LIN {X 0,Y 607.534,Z 521.411,A -85,B 0,C 180,E1 27658.35,E2 27658.35} C_VEL
LIN {X 0,Y 606.937,Z 539.809,A -85,B 0,C 180,E1 27658.034,E2 27658.034} C_VEL
LIN {X 0,Y 606.179,Z 557.221,A -85,B 0,C 180,E1 27657.624,E2 27657.624} C_VEL
LIN {X 0,Y 605.306,Z 574.046,A -85,B 0,C 180,E1 27657.12,E2 27657.12} C_VEL
LIN {X 0,Y 604.323,Z 590.19,A -85,B 0,C 180,E1 27656.53,E2 27656.53} C_VEL
LIN {X 0,Y 603.193,Z 607.046,A -85,B 0,C 180,E1 27655.795,E2 27655.795} C_VEL
LIN {X 0,Y 601.778,Z 626.286,A -85,B 0,C 180,E1 27654.802,E2 27654.802} C_VEL
LIN {X 0,Y 600.164,Z 646.019,A -85,B 0,C 180,E1 27653.565,E2 27653.565} C_VEL
LIN {X 0,Y 598.909,Z 660.987,A -85,B 0,C 180,E1 27652.474,E2 27652.474} C_VEL
LIN {X 0,Y 597.728,Z 674.768,A -85,B 0,C 180,E1 27651.333,E2 27651.333} C_VEL
LIN {X 0,Y 596.656,Z 687.506,A -85,B 0,C 180,E1 27650.141,E2 27650.141} C_VEL
LIN {X 0,Y 595.699,Z 699.296,A -85,B 0,C 180,E1 27648.899,E2 27648.899} C_VEL
LIN {X 0,Y 594.784,Z 710.992,A -85,B 0,C 180,E1 27647.51,E2 27647.51} C_VEL
LIN {X 0,Y 593.947,Z 722.712,A -85,B 0,C 180,E1 27645.924,E2 27645.924} C_VEL
LIN {X 0,Y 593.118,Z 735.863,A -85,B 0,C 180,E1 27643.823,E2 27643.823} C_VEL
LIN {X 0,Y 592.654,Z 744.533,A -85,B 0,C 180,E1 27642.173,E2 27642.173} C_VEL
LIN {X 0,Y 592.352,Z 751.606,A -85,B 0,C 180,E1 27640.601,E2 27640.601} C_VEL
LIN {X 0,Y 592.127,Z 757.906,A -85,B 0,C 180,E1 27638.936,E2 27638.936} C_VEL
LIN {X 0,Y 592.011,Z 763.04,A -85,B 0,C 180,E1 27637.276,E2 27637.276} C_VEL
LIN {X 0,Y 591.947,Z 767.067,A -85,B 0,C 180,E1 27635.622,E2 27635.622} C_VEL
LIN {X 0,Y 591.925,Z 770.029,A -85,B 0,C 180,E1 27633.971,E2 27633.971} C_VEL
LIN {X 0,Y 591.913,Z 772.046,A -85,B 0,C 180,E1 27632.226,E2 27632.226} C_VEL
LIN {X 0,Y 591.908,Z 772.99,A -85,B 0,C 180,E1 27630.29,E2 27630.29} C_VEL
LIN {X 0,Y 591.917,Z 772.222,A -85,B 0,C 180,E1 27627.967,E2 27627.967} C_VEL
LIN {X 0,Y 591.924,Z 770.176,A -85,B 0,C 180,E1 27626.126,E2 27626.126} C_VEL
LIN {X 0,Y 591.944,Z 767.274,A -85,B 0,C 180,E1 27624.476,E2 27624.476} C_VEL
LIN {X 0,Y 592.002,Z 763.31,A -85,B 0,C 180,E1 27622.821,E2 27622.821} C_VEL
LIN {X 0,Y 592.116,Z 758.239,A -85,B 0,C 180,E1 27621.162,E2 27621.162} C_VEL
LIN {X 0,Y 592.323,Z 752.405,A -85,B 0,C 180,E1 27619.595,E2 27619.595} C_VEL
LIN {X 0,Y 592.61,Z 745.469,A -85,B 0,C 180,E1 27618.024,E2 27618.024} C_VEL
LIN {X 0,Y 593.024,Z 737.35,A -85,B 0,C 180,E1 27616.448,E2 27616.448} C_VEL
LIN {X 0,Y 593.643,Z 727.32,A -85,B 0,C 180,E1 27614.769,E2 27614.769} C_VEL
LIN {X 0,Y 594.627,Z 713.225,A -85,B 0,C 180,E1 27612.77,E2 27612.77} C_VEL
LIN {X 0,Y 595.607,Z 700.484,A -85,B 0,C 180,E1 27611.233,E2 27611.233} C_VEL
LIN {X 0,Y 596.616,Z 688.006,A -85,B 0,C 180,E1 27609.909,E2 27609.909} C_VEL
LIN {X 0,Y 597.677,Z 675.329,A -85,B 0,C 180,E1 27608.717,E2 27608.717} C_VEL
LIN {X 0,Y 598.853,Z 661.617,A -85,B 0,C 180,E1 27607.575,E2 27607.575} C_VEL
LIN {X 0,Y 600.104,Z 646.73,A -85,B 0,C 180,E1 27606.484,E2 27606.484} C_VEL
LIN {X 0,Y 601.642,Z 628.036,A -85,B 0,C 180,E1 27605.297,E2 27605.297} C_VEL
LIN {X 0,Y 603.118,Z 608.215,A -85,B 0,C 180,E1 27604.259,E2 27604.259} C_VEL
LIN {X 0,Y 604.251,Z 591.435,A -85,B 0,C 180,E1 27603.519,E2 27603.519} C_VEL
LIN {X 0,Y 605.262,Z 574.876,A -85,B 0,C 180,E1 27602.908,E2 27602.908} C_VEL
LIN {X 0,Y 606.173,Z 557.347,A -85,B 0,C 180,E1 27602.379,E2 27602.379} C_VEL
LIN {X 0,Y 606.929,Z 539.917,A -85,B 0,C 180,E1 27601.968,E2 27601.968} C_VEL
LIN {X 0,Y 607.522,Z 521.806,A -85,B 0,C 180,E1 27601.656,E2 27601.656} C_VEL
LIN {X 0,Y 611.396,Z 259.873,A -85,B 0,C 180,E1 27598.361,E2 27598.361} C_VEL
LIN {X 0,Y 611.12,Z 255.681,A -85,B 0,C 180,E1 27598.289,E2 27598.289} C_VEL
LIN {X 0,Y 604.007,Z 223.457,A -85,B 0,C 180,E1 27597.418,E2 27597.418} C_VEL
LIN {X 0,Y 601.164,Z 213.241,A -85,B 0,C 180,E1 27596.258,E2 27596.258} C_VEL
LIN {X 0,Y 594.896,Z 192.872,A -85,B 0,C 180,E1 27593.782,E2 27593.782} C_VEL
LIN {X 0,Y 593.129,Z 187.4,A -85,B 0,C 180,E1 27593.041,E2 27593.041} C_VEL
LIN {X 0,Y 593.122,Z 187.284,A -85,B 0,C 180,E1 27589.917,E2 27589.917} C_VEL
LIN {X 0,Y 593.118,Z 187.278,A -85,B 0,C 180,E1 27587.025,E2 27587.025} C_VEL
LIN {X 0,Y 593.105,Z 187.276,A -85,B 0,C 180,E1 27583.726,E2 27583.726} C_VEL
LIN {X 0,Y 593.165,Z 187.265,A -85,B 0,C 180,E1 27580.672,E2 27580.672} C_VEL
LIN {X 0,Y 593.102,Z 187.286,A -85,B 0,C 180,E1 27577.604,E2 27577.604} C_VEL
LIN {X 0,Y 593.164,Z 187.259,A -85,B 0,C 180,E1 27574.494,E2 27574.494} C_VEL
LIN {X 0,Y 593.104,Z 187.285,A -85,B 0,C 180,E1 27571.468,E2 27571.468} C_VEL
LIN {X 0,Y 593.129,Z 187.242,A -85,B 0,C 180,E1 27568.275,E2 27568.275} C_VEL
LIN {X 0,Y 593.113,Z 187.278,A -85,B 0,C 180,E1 27565.354,E2 27565.354} C_VEL
LIN {X 0,Y 593.109,Z 187.274,A -85,B 0,C 180,E1 27562.083,E2 27562.083} C_VEL
LIN {X 0,Y 593.131,Z 187.283,A -85,B 0,C 180,E1 27559.192,E2 27559.192} C_VEL
LIN {X 0,Y 593.106,Z 187.282,A -85,B 0,C 180,E1 27556.05,E2 27556.05} C_VEL
LIN {X 0,Y 593.141,Z 187.272,A -85,B 0,C 180,E1 27553.155,E2 27553.155} C_VEL
LIN {X 0,Y 593.102,Z 187.282,A -85,B 0,C 180,E1 27550,E2 27550} C_VEL
LIN {X 0,Y 593.178,Z 187.272,A -85,B 0,C 180,E1 27546.874,E2 27546.874} C_VEL
LIN {X 0,Y 593.101,Z 187.279,A -85,B 0,C 180,E1 27543.77,E2 27543.77} C_VEL
LIN {X 0,Y 593.129,Z 187.285,A -85,B 0,C 180,E1 27540.58,E2 27540.58} C_VEL
LIN {X 0,Y 593.107,Z 187.271,A -85,B 0,C 180,E1 27537.681,E2 27537.681} C_VEL
LIN {X 0,Y 593.108,Z 187.281,A -85,B 0,C 180,E1 27534.389,E2 27534.389} C_VEL
LIN {X 0,Y 593.122,Z 187.277,A -85,B 0,C 180,E1 27531.566,E2 27531.566} C_VEL
LIN {X 0,Y 593.102,Z 187.274,A -85,B 0,C 180,E1 27528.328,E2 27528.328} C_VEL
LIN {X 0,Y 593.169,Z 187.284,A -85,B 0,C 180,E1 27525.254,E2 27525.254} C_VEL
LIN {X 0,Y 593.101,Z 187.279,A -85,B 0,C 180,E1 27522.132,E2 27522.132} C_VEL
LIN {X 0,Y 593.154,Z 187.272,A -85,B 0,C 180,E1 27519.028,E2 27519.028} C_VEL
LIN {X 0,Y 593.102,Z 187.285,A -85,B 0,C 180,E1 27516.133,E2 27516.133} C_VEL
LIN {X 0,Y 593.144,Z 187.24,A -85,B 0,C 180,E1 27513.034,E2 27513.034} C_VEL
LIN {X 0,Y 593.105,Z 187.274,A -85,B 0,C 180,E1 27510.044,E2 27510.044} C_VEL
LIN {X 0,Y 593.11,Z 187.273,A -85,B 0,C 180,E1 27506.727,E2 27506.727} C_VEL
LIN {X 0,Y 593.135,Z 187.257,A -85,B 0,C 180,E1 27503.722,E2 27503.722} C_VEL
LIN {X 0,Y 593.104,Z 187.286,A -85,B 0,C 180,E1 27500.663,E2 27500.663} C_VEL
LIN {X 0,Y 593.148,Z 187.286,A -85,B 0,C 180,E1 27497.726,E2 27497.726} C_VEL
LIN {X 0,Y 593.101,Z 187.287,A -85,B 0,C 180,E1 27494.648,E2 27494.648} C_VEL
LIN {X 0,Y 593.18,Z 187.282,A -85,B 0,C 180,E1 27491.545,E2 27491.545} C_VEL
LIN {X 0,Y 593.099,Z 187.287,A -85,B 0,C 180,E1 27488.533,E2 27488.533} C_VEL
LIN {X 0,Y 593.16,Z 187.283,A -85,B 0,C 180,E1 27485.437,E2 27485.437} C_VEL
LIN {X 0,Y 593.104,Z 187.288,A -85,B 0,C 180,E1 27482.414,E2 27482.414} C_VEL
LIN {X 0,Y 593.12,Z 187.288,A -85,B 0,C 180,E1 27479.152,E2 27479.152} C_VEL
LIN {X 0,Y 593.123,Z 187.285,A -85,B 0,C 180,E1 27476.207,E2 27476.207} C_VEL
LIN {X 0,Y 593.105,Z 187.288,A -85,B 0,C 180,E1 27474.901,E2 27474.901} C_VEL
LIN {X 0,Y 592.123,Z 187.413,A -85,B 0,C 180,E1 27474.158,E2 27474.158} C_VEL
LIN {X 0,Y 585.692,Z 188.216,A -85,B 0,C 180,E1 27472.015,E2 27472.015} C_VEL
LIN {X 0,Y 585.212,Z 188.273,A -85,B 0,C 180,E1 27471.526,E2 27471.526} C_VEL
LIN {X 0,Y 585.169,Z 188.277,A -85,B 0,C 180,E1 27468.496,E2 27468.496} C_VEL
LIN {X 0,Y 585.169,Z 188.279,A -85,B 0,C 180,E1 27465.153,E2 27465.153} C_VEL
LIN {X 0,Y 585.197,Z 188.276,A -85,B 0,C 180,E1 27462.219,E2 27462.219} C_VEL
LIN {X 0,Y 585.16,Z 188.277,A -85,B 0,C 180,E1 27459.011,E2 27459.011} C_VEL
LIN {X 0,Y 585.234,Z 188.269,A -85,B 0,C 180,E1 27455.981,E2 27455.981} C_VEL
LIN {X 0,Y 585.161,Z 188.279,A -85,B 0,C 180,E1 27452.84,E2 27452.84} C_VEL
LIN {X 0,Y 585.19,Z 188.274,A -85,B 0,C 180,E1 27449.608,E2 27449.608} C_VEL
LIN {X 0,Y 585.171,Z 188.276,A -85,B 0,C 180,E1 27446.67,E2 27446.67} C_VEL
LIN {X 0,Y 585.166,Z 188.28,A -85,B 0,C 180,E1 27443.328,E2 27443.328} C_VEL
LIN {X 0,Y 585.208,Z 188.275,A -85,B 0,C 180,E1 27440.357,E2 27440.357} C_VEL
LIN {X 0,Y 585.161,Z 188.276,A -85,B 0,C 180,E1 27437.268,E2 27437.268} C_VEL
LIN {X 0,Y 585.233,Z 188.27,A -85,B 0,C 180,E1 27434.239,E2 27434.239} C_VEL
LIN {X 0,Y 585.162,Z 188.278,A -85,B 0,C 180,E1 27431.161,E2 27431.161} C_VEL
LIN {X 0,Y 585.213,Z 188.273,A -85,B 0,C 180,E1 27428.029,E2 27428.029} C_VEL
LIN {X 0,Y 585.168,Z 188.278,A -85,B 0,C 180,E1 27425.039,E2 27425.039} C_VEL
LIN {X 0,Y 585.177,Z 188.277,A -85,B 0,C 180,E1 27421.755,E2 27421.755} C_VEL
LIN {X 0,Y 585.185,Z 188.274,A -85,B 0,C 180,E1 27418.825,E2 27418.825} C_VEL
LIN {X 0,Y 585.164,Z 188.277,A -85,B 0,C 180,E1 27415.562,E2 27415.562} C_VEL
LIN {X 0,Y 585.234,Z 188.271,A -85,B 0,C 180,E1 27412.421,E2 27412.421} C_VEL
LIN {X 0,Y 585.163,Z 188.275,A -85,B 0,C 180,E1 27409.348,E2 27409.348} C_VEL
LIN {X 0,Y 585.207,Z 188.274,A -85,B 0,C 180,E1 27406.22,E2 27406.22} C_VEL
LIN {X 0,Y 585.173,Z 188.276,A -85,B 0,C 180,E1 27403.154,E2 27403.154} C_VEL
LIN {X 0,Y 585.168,Z 188.275,A -85,B 0,C 180,E1 27399.85,E2 27399.85} C_VEL
LIN {X 0,Y 585.198,Z 188.259,A -85,B 0,C 180,E1 27396.915,E2 27396.915} C_VEL
LIN {X 0,Y 585.16,Z 188.26,A -85,B 0,C 180,E1 27393.734,E2 27393.734} C_VEL
LIN {X 0,Y 585.239,Z 188.262,A -85,B 0,C 180,E1 27390.607,E2 27390.607} C_VEL
LIN {X 0,Y 585.16,Z 188.225,A -85,B 0,C 180,E1 27387.475,E2 27387.475} C_VEL
LIN {X 0,Y 585.178,Z 188.274,A -85,B 0,C 180,E1 27384.173,E2 27384.173} C_VEL
LIN {X 0,Y 585.177,Z 188.262,A -85,B 0,C 180,E1 27381.343,E2 27381.343} C_VEL
LIN {X 0,Y 585.17,Z 188.267,A -85,B 0,C 180,E1 27378.119,E2 27378.119} C_VEL
LIN {X 0,Y 585.212,Z 188.269,A -85,B 0,C 180,E1 27375.053,E2 27375.053} C_VEL
LIN {X 0,Y 585.16,Z 188.261,A -85,B 0,C 180,E1 27371.932,E2 27371.932} C_VEL
LIN {X 0,Y 585.231,Z 188.265,A -85,B 0,C 180,E1 27368.845,E2 27368.845} C_VEL
LIN {X 0,Y 585.163,Z 188.27,A -85,B 0,C 180,E1 27365.786,E2 27365.786} C_VEL
LIN {X 0,Y 585.187,Z 188.258,A -85,B 0,C 180,E1 27362.546,E2 27362.546} C_VEL
LIN {X 0,Y 585.174,Z 188.273,A -85,B 0,C 180,E1 27359.608,E2 27359.608} C_VEL
LIN {X 0,Y 585.164,Z 188.266,A -85,B 0,C 180,E1 27356.277,E2 27356.277} C_VEL
LIN {X 0,Y 585.237,Z 188.259,A -85,B 0,C 180,E1 27353.131,E2 27353.131} C_VEL
LIN {X 0,Y 585.162,Z 188.271,A -85,B 0,C 180,E1 27350.062,E2 27350.062} C_VEL
LIN {X 0,Y 585.204,Z 188.262,A -85,B 0,C 180,E1 27346.85,E2 27346.85} C_VEL
LIN {X 0,Y 585.168,Z 188.273,A -85,B 0,C 180,E1 27343.93,E2 27343.93} C_VEL
LIN {X 0,Y 585.173,Z 188.274,A -85,B 0,C 180,E1 27340.575,E2 27340.575} C_VEL
LIN {X 0,Y 585.203,Z 188.261,A -85,B 0,C 180,E1 27337.553,E2 27337.553} C_VEL
LIN {X 0,Y 585.164,Z 188.267,A -85,B 0,C 180,E1 27334.386,E2 27334.386} C_VEL
LIN {X 0,Y 585.234,Z 188.225,A -85,B 0,C 180,E1 27331.308,E2 27331.308} C_VEL
LIN {X 0,Y 585.165,Z 188.274,A -85,B 0,C 180,E1 27328.245,E2 27328.245} C_VEL
LIN {X 0,Y 585.2,Z 188.248,A -85,B 0,C 180,E1 27325.083,E2 27325.083} C_VEL
LIN {X 0,Y 585.177,Z 188.275,A -85,B 0,C 180,E1 27322.038,E2 27322.038} C_VEL
LIN {X 0,Y 585.169,Z 188.272,A -85,B 0,C 180,E1 27318.733,E2 27318.733} C_VEL
LIN {X 0,Y 585.219,Z 188.253,A -85,B 0,C 180,E1 27315.668,E2 27315.668} C_VEL
LIN {X 0,Y 585.162,Z 188.264,A -85,B 0,C 180,E1 27312.568,E2 27312.568} C_VEL
LIN {X 0,Y 585.224,Z 188.243,A -85,B 0,C 180,E1 27309.442,E2 27309.442} C_VEL
LIN {X 0,Y 585.241,Z 188.445,A -85,B 0,C 180,E1 27307.383,E2 27307.383} C_VEL
LIN {X 0,Y 591.021,Z 206.75,A -85,B 0,C 180,E1 27305.032,E2 27305.032} C_VEL
LIN {X 0,Y 595.736,Z 222.647,A -85,B 0,C 180,E1 27303.12,E2 27303.12} C_VEL
LIN {X 0,Y 597.814,Z 227.828,A -85,B 0,C 180,E1 27302.887,E2 27302.887} C_VEL
LIN {X 0,Y 604.586,Z 259.317,A -85,B 0,C 180,E1 27302.043,E2 27302.043} C_VEL
LIN {X 0,Y 600.477,Z 521.632,A -85,B 0,C 180,E1 27298.707,E2 27298.707} C_VEL
LIN {X 0,Y 599.862,Z 539.666,A -85,B 0,C 180,E1 27298.393,E2 27298.393} C_VEL
LIN {X 0,Y 599.065,Z 557.04,A -85,B 0,C 180,E1 27297.981,E2 27297.981} C_VEL
LIN {X 0,Y 598.143,Z 573.87,A -85,B 0,C 180,E1 27297.472,E2 27297.472} C_VEL
LIN {X 0,Y 597.105,Z 590.013,A -85,B 0,C 180,E1 27296.877,E2 27296.877} C_VEL
LIN {X 0,Y 595.904,Z 606.974,A -85,B 0,C 180,E1 27296.129,E2 27296.129} C_VEL
LIN {X 0,Y 594.351,Z 627.019,A -85,B 0,C 180,E1 27295.08,E2 27295.08} C_VEL
LIN {X 0,Y 592.707,Z 645.841,A -85,B 0,C 180,E1 27293.88,E2 27293.88} C_VEL
LIN {X 0,Y 591.379,Z 660.809,A -85,B 0,C 180,E1 27292.776,E2 27292.776} C_VEL
LIN {X 0,Y 590.131,Z 674.59,A -85,B 0,C 180,E1 27291.621,E2 27291.621} C_VEL
LIN {X 0,Y 589,Z 687.154,A -85,B 0,C 180,E1 27290.432,E2 27290.432} C_VEL
LIN {X 0,Y 587.963,Z 699.117,A -85,B 0,C 180,E1 27289.158,E2 27289.158} C_VEL
LIN {X 0,Y 586.992,Z 710.813,A -85,B 0,C 180,E1 27287.75,E2 27287.75} C_VEL
LIN {X 0,Y 586.094,Z 722.533,A -85,B 0,C 180,E1 27286.143,E2 27286.143} C_VEL
LIN {X 0,Y 585.211,Z 735.548,A -85,B 0,C 180,E1 27284.039,E2 27284.039} C_VEL
LIN {X 0,Y 584.705,Z 744.355,A -85,B 0,C 180,E1 27282.341,E2 27282.341} C_VEL
LIN {X 0,Y 584.382,Z 751.429,A -85,B 0,C 180,E1 27280.747,E2 27280.747} C_VEL
LIN {X 0,Y 584.148,Z 757.73,A -85,B 0,C 180,E1 27279.059,E2 27279.059} C_VEL
LIN {X 0,Y 584.022,Z 762.595,A -85,B 0,C 180,E1 27277.475,E2 27277.475} C_VEL
LIN {X 0,Y 583.952,Z 766.683,A -85,B 0,C 180,E1 27275.797,E2 27275.797} C_VEL
LIN {X 0,Y 583.926,Z 769.706,A -85,B 0,C 180,E1 27274.124,E2 27274.124} C_VEL
LIN {X 0,Y 583.915,Z 771.695,A -85,B 0,C 180,E1 27272.453,E2 27272.453} C_VEL
LIN {X 0,Y 583.914,Z 772.67,A -85,B 0,C 180,E1 27270.785,E2 27270.785} C_VEL
LIN {X 0,Y 583.915,Z 772.64,A -85,B 0,C 180,E1 27269.117,E2 27269.117} C_VEL
LIN {X 0,Y 583.916,Z 771.607,A -85,B 0,C 180,E1 27267.449,E2 27267.449} C_VEL
LIN {X 0,Y 583.926,Z 769.559,A -85,B 0,C 180,E1 27265.778,E2 27265.778} C_VEL
LIN {X 0,Y 583.961,Z 766.268,A -85,B 0,C 180,E1 27264.005,E2 27264.005} C_VEL
LIN {X 0,Y 584.051,Z 761.247,A -85,B 0,C 180,E1 27262.03,E2 27262.03} C_VEL
LIN {X 0,Y 584.288,Z 753.824,A -85,B 0,C 180,E1 27259.849,E2 27259.849} C_VEL
LIN {X 0,Y 584.616,Z 746.178,A -85,B 0,C 180,E1 27258.047,E2 27258.047} C_VEL
LIN {X 0,Y 585.039,Z 738.254,A -85,B 0,C 180,E1 27256.461,E2 27256.461} C_VEL
LIN {X 0,Y 585.597,Z 729.616,A -85,B 0,C 180,E1 27254.96,E2 27254.96} C_VEL
LIN {X 0,Y 586.294,Z 719.727,A -85,B 0,C 180,E1 27253.455,E2 27253.455} C_VEL
LIN {X 0,Y 587.189,Z 708.438,A -85,B 0,C 180,E1 27251.948,E2 27251.948} C_VEL
LIN {X 0,Y 588.456,Z 693.775,A -85,B 0,C 180,E1 27250.239,E2 27250.239} C_VEL
LIN {X 0,Y 589.877,Z 677.395,A -85,B 0,C 180,E1 27248.63,E2 27248.63} C_VEL
LIN {X 0,Y 591.151,Z 663.331,A -85,B 0,C 180,E1 27247.424,E2 27247.424} C_VEL
LIN {X 0,Y 592.396,Z 649.397,A -85,B 0,C 180,E1 27246.371,E2 27246.371} C_VEL
LIN {X 0,Y 593.634,Z 635.116,A -85,B 0,C 180,E1 27245.419,E2 27245.419} C_VEL
LIN {X 0,Y 594.895,Z 619.661,A -85,B 0,C 180,E1 27244.518,E2 27244.518} C_VEL
LIN {X 0,Y 596.132,Z 603.786,A -85,B 0,C 180,E1 27243.721,E2 27243.721} C_VEL
LIN {X 0,Y 597.364,Z 586.279,A -85,B 0,C 180,E1 27242.975,E2 27242.975} C_VEL
LIN {X 0,Y 598.743,Z 564.3,A -85,B 0,C 180,E1 27242.217,E2 27242.217} C_VEL
LIN {X 0,Y 599.718,Z 542.973,A -85,B 0,C 180,E1 27241.675,E2 27241.675} C_VEL
LIN {X 0,Y 600.382,Z 524.916,A -85,B 0,C 180,E1 27241.342,E2 27241.342} C_VEL
LIN {X 0,Y 603.434,Z 330.012,A -85,B 0,C 180,E1 27238.856,E2 27238.856} C_VEL
LIN {X 0,Y 604.421,Z 257.818,A -85,B 0,C 180,E1 27237.927,E2 27237.927} C_VEL
LIN {X 0,Y 597.247,Z 226.077,A -85,B 0,C 180,E1 27237.054,E2 27237.054} C_VEL
LIN {X 0,Y 595.679,Z 222.484,A -85,B 0,C 180,E1 27236.867,E2 27236.867} C_VEL
LIN {X 0,Y 590.094,Z 203.733,A -85,B 0,C 180,E1 27234.59,E2 27234.59} C_VEL
LIN {X 0,Y 585.237,Z 188.416,A -85,B 0,C 180,E1 27232.605,E2 27232.605} C_VEL
LIN {X 0,Y 585.165,Z 188.28,A -85,B 0,C 180,E1 27229.499,E2 27229.499} C_VEL
LIN {X 0,Y 585.232,Z 188.27,A -85,B 0,C 180,E1 27226.421,E2 27226.421} C_VEL
LIN {X 0,Y 585.169,Z 188.268,A -85,B 0,C 180,E1 27223.251,E2 27223.251} C_VEL
LIN {X 0,Y 585.172,Z 188.255,A -85,B 0,C 180,E1 27219.905,E2 27219.905} C_VEL
LIN {X 0,Y 585.184,Z 188.275,A -85,B 0,C 180,E1 27217.076,E2 27217.076} C_VEL
LIN {X 0,Y 585.167,Z 188.265,A -85,B 0,C 180,E1 27213.852,E2 27213.852} C_VEL
LIN {X 0,Y 585.228,Z 188.26,A -85,B 0,C 180,E1 27210.764,E2 27210.764} C_VEL
LIN {X 0,Y 585.158,Z 188.236,A -85,B 0,C 180,E1 27207.696,E2 27207.696} C_VEL
LIN {X 0,Y 585.218,Z 188.274,A -85,B 0,C 180,E1 27204.531,E2 27204.531} C_VEL
LIN {X 0,Y 585.163,Z 188.263,A -85,B 0,C 180,E1 27201.554,E2 27201.554} C_VEL
LIN {X 0,Y 585.187,Z 188.26,A -85,B 0,C 180,E1 27198.324,E2 27198.324} C_VEL
LIN {X 0,Y 585.181,Z 188.271,A -85,B 0,C 180,E1 27195.358,E2 27195.358} C_VEL
LIN {X 0,Y 585.168,Z 188.267,A -85,B 0,C 180,E1 27192.133,E2 27192.133} C_VEL
LIN {X 0,Y 585.222,Z 188.263,A -85,B 0,C 180,E1 27189.044,E2 27189.044} C_VEL
LIN {X 0,Y 585.162,Z 188.273,A -85,B 0,C 180,E1 27185.983,E2 27185.983} C_VEL
LIN {X 0,Y 585.222,Z 188.258,A -85,B 0,C 180,E1 27182.84,E2 27182.84} C_VEL
LIN {X 0,Y 585.164,Z 188.273,A -85,B 0,C 180,E1 27179.804,E2 27179.804} C_VEL
LIN {X 0,Y 585.186,Z 188.272,A -85,B 0,C 180,E1 27176.571,E2 27176.571} C_VEL
LIN {X 0,Y 585.177,Z 188.27,A -85,B 0,C 180,E1 27173.623,E2 27173.623} C_VEL
LIN {X 0,Y 585.166,Z 188.274,A -85,B 0,C 180,E1 27170.333,E2 27170.333} C_VEL
LIN {X 0,Y 585.232,Z 188.258,A -85,B 0,C 180,E1 27167.167,E2 27167.167} C_VEL
LIN {X 0,Y 585.16,Z 188.27,A -85,B 0,C 180,E1 27164.132,E2 27164.132} C_VEL
LIN {X 0,Y 585.211,Z 188.273,A -85,B 0,C 180,E1 27160.953,E2 27160.953} C_VEL
LIN {X 0,Y 585.169,Z 188.264,A -85,B 0,C 180,E1 27157.919,E2 27157.919} C_VEL
LIN {X 0,Y 585.171,Z 188.262,A -85,B 0,C 180,E1 27154.603,E2 27154.603} C_VEL
LIN {X 0,Y 585.211,Z 188.225,A -85,B 0,C 180,E1 27151.53,E2 27151.53} C_VEL
LIN {X 0,Y 585.164,Z 188.275,A -85,B 0,C 180,E1 27148.475,E2 27148.475} C_VEL
LIN {X 0,Y 585.225,Z 188.234,A -85,B 0,C 180,E1 27145.428,E2 27145.428} C_VEL
LIN {X 0,Y 585.163,Z 188.273,A -85,B 0,C 180,E1 27142.283,E2 27142.283} C_VEL
LIN {X 0,Y 585.201,Z 188.275,A -85,B 0,C 180,E1 27139.125,E2 27139.125} C_VEL
LIN {X 0,Y 585.176,Z 188.275,A -85,B 0,C 180,E1 27136.074,E2 27136.074} C_VEL
LIN {X 0,Y 585.17,Z 188.276,A -85,B 0,C 180,E1 27132.842,E2 27132.842} C_VEL
LIN {X 0,Y 585.198,Z 188.275,A -85,B 0,C 180,E1 27129.899,E2 27129.899} C_VEL
LIN {X 0,Y 585.164,Z 188.275,A -85,B 0,C 180,E1 27126.725,E2 27126.725} C_VEL
LIN {X 0,Y 585.234,Z 188.27,A -85,B 0,C 180,E1 27123.607,E2 27123.607} C_VEL
LIN {X 0,Y 585.163,Z 188.275,A -85,B 0,C 180,E1 27120.492,E2 27120.492} C_VEL
LIN {X 0,Y 585.195,Z 188.275,A -85,B 0,C 180,E1 27117.315,E2 27117.315} C_VEL
LIN {X 0,Y 585.177,Z 188.278,A -85,B 0,C 180,E1 27114.314,E2 27114.314} C_VEL
LIN {X 0,Y 585.212,Z 188.273,A -85,B 0,C 180,E1 27111.526,E2 27111.526} C_VEL
LIN {X 0,Y 584.146,Z 188.404,A -85,B 0,C 180,E1 27110.772,E2 27110.772} C_VEL
LIN {X 0,Y 577.743,Z 189.203,A -85,B 0,C 180,E1 27108.656,E2 27108.656} C_VEL
LIN {X 0,Y 577.264,Z 189.262,A -85,B 0,C 180,E1 27108.105,E2 27108.105} C_VEL
LIN {X 0,Y 577.223,Z 189.268,A -85,B 0,C 180,E1 27104.956,E2 27104.956} C_VEL
LIN {X 0,Y 577.29,Z 189.26,A -85,B 0,C 180,E1 27101.873,E2 27101.873} C_VEL
LIN {X 0,Y 577.222,Z 189.265,A -85,B 0,C 180,E1 27098.767,E2 27098.767} C_VEL
LIN {X 0,Y 577.255,Z 189.266,A -85,B 0,C 180,E1 27095.566,E2 27095.566} C_VEL
LIN {X 0,Y 577.242,Z 189.267,A -85,B 0,C 180,E1 27092.482,E2 27092.482} C_VEL
LIN {X 0,Y 577.23,Z 189.265,A -85,B 0,C 180,E1 27089.305,E2 27089.305} C_VEL
LIN {X 0,Y 577.275,Z 189.261,A -85,B 0,C 180,E1 27086.227,E2 27086.227} C_VEL
LIN {X 0,Y 577.223,Z 189.269,A -85,B 0,C 180,E1 27083.136,E2 27083.136} C_VEL
LIN {X 0,Y 577.287,Z 189.259,A -85,B 0,C 180,E1 27080.027,E2 27080.027} C_VEL
LIN {X 0,Y 577.229,Z 189.264,A -85,B 0,C 180,E1 27076.886,E2 27076.886} C_VEL
LIN {X 0,Y 577.232,Z 189.266,A -85,B 0,C 180,E1 27073.498,E2 27073.498} C_VEL
LIN {X 0,Y 577.283,Z 189.26,A -85,B 0,C 180,E1 27070.368,E2 27070.368} C_VEL
LIN {X 0,Y 577.223,Z 189.266,A -85,B 0,C 180,E1 27067.279,E2 27067.279} C_VEL
LIN {X 0,Y 577.282,Z 189.263,A -85,B 0,C 180,E1 27064.124,E2 27064.124} C_VEL
LIN {X 0,Y 577.231,Z 189.267,A -85,B 0,C 180,E1 27061.018,E2 27061.018} C_VEL
LIN {X 0,Y 577.229,Z 189.266,A -85,B 0,C 180,E1 27057.644,E2 27057.644} C_VEL
LIN {X 0,Y 577.283,Z 189.261,A -85,B 0,C 180,E1 27054.538,E2 27054.538} C_VEL
LIN {X 0,Y 577.222,Z 189.266,A -85,B 0,C 180,E1 27051.375,E2 27051.375} C_VEL
LIN {X 0,Y 577.281,Z 189.261,A -85,B 0,C 180,E1 27048.29,E2 27048.29} C_VEL
LIN {X 0,Y 577.231,Z 189.265,A -85,B 0,C 180,E1 27045.177,E2 27045.177} C_VEL
LIN {X 0,Y 577.231,Z 189.264,A -85,B 0,C 180,E1 27041.829,E2 27041.829} C_VEL
LIN {X 0,Y 577.274,Z 189.263,A -85,B 0,C 180,E1 27038.8,E2 27038.8} C_VEL
LIN {X 0,Y 577.217,Z 189.229,A -85,B 0,C 180,E1 27035.677,E2 27035.677} C_VEL
LIN {X 0,Y 577.28,Z 189.257,A -85,B 0,C 180,E1 27032.476,E2 27032.476} C_VEL
LIN {X 0,Y 577.223,Z 189.244,A -85,B 0,C 180,E1 27029.469,E2 27029.469} C_VEL
LIN {X 0,Y 577.242,Z 189.235,A -85,B 0,C 180,E1 27026.213,E2 27026.213} C_VEL
LIN {X 0,Y 577.253,Z 189.263,A -85,B 0,C 180,E1 27023.154,E2 27023.154} C_VEL
LIN {X 0,Y 577.225,Z 189.262,A -85,B 0,C 180,E1 27019.953,E2 27019.953} C_VEL
LIN {X 0,Y 577.292,Z 189.246,A -85,B 0,C 180,E1 27016.813,E2 27016.813} C_VEL
LIN {X 0,Y 577.222,Z 189.26,A -85,B 0,C 180,E1 27013.728,E2 27013.728} C_VEL
LIN {X 0,Y 577.252,Z 189.262,A -85,B 0,C 180,E1 27010.479,E2 27010.479} C_VEL
LIN {X 0,Y 577.24,Z 189.251,A -85,B 0,C 180,E1 27007.465,E2 27007.465} C_VEL
LIN {X 0,Y 577.225,Z 189.261,A -85,B 0,C 180,E1 27004.172,E2 27004.172} C_VEL
LIN {X 0,Y 577.296,Z 189.249,A -85,B 0,C 180,E1 27000.992,E2 27000.992} C_VEL
LIN {X 0,Y 577.223,Z 189.255,A -85,B 0,C 180,E1 26997.915,E2 26997.915} C_VEL
LIN {X 0,Y 577.261,Z 189.26,A -85,B 0,C 180,E1 26994.733,E2 26994.733} C_VEL
LIN {X 0,Y 577.232,Z 189.245,A -85,B 0,C 180,E1 26991.734,E2 26991.734} C_VEL
LIN {X 0,Y 577.229,Z 189.256,A -85,B 0,C 180,E1 26988.408,E2 26988.408} C_VEL
LIN {X 0,Y 577.295,Z 189.257,A -85,B 0,C 180,E1 26985.25,E2 26985.25} C_VEL
LIN {X 0,Y 577.224,Z 189.25,A -85,B 0,C 180,E1 26982.145,E2 26982.145} C_VEL
LIN {X 0,Y 577.27,Z 189.253,A -85,B 0,C 180,E1 26978.983,E2 26978.983} C_VEL
LIN {X 0,Y 577.233,Z 189.262,A -85,B 0,C 180,E1 26975.979,E2 26975.979} C_VEL
LIN {X 0,Y 577.232,Z 189.226,A -85,B 0,C 180,E1 26972.675,E2 26972.675} C_VEL
LIN {X 0,Y 577.268,Z 189.243,A -85,B 0,C 180,E1 26969.617,E2 26969.617} C_VEL
LIN {X 0,Y 577.223,Z 189.255,A -85,B 0,C 180,E1 26966.455,E2 26966.455} C_VEL
LIN {X 0,Y 577.286,Z 189.253,A -85,B 0,C 180,E1 26963.305,E2 26963.305} C_VEL
LIN {X 0,Y 577.224,Z 189.245,A -85,B 0,C 180,E1 26960.265,E2 26960.265} C_VEL
LIN {X 0,Y 577.256,Z 189.257,A -85,B 0,C 180,E1 26957.099,E2 26957.099} C_VEL
LIN {X 0,Y 577.245,Z 189.263,A -85,B 0,C 180,E1 26954.04,E2 26954.04} C_VEL
LIN {X 0,Y 577.23,Z 189.269,A -85,B 0,C 180,E1 26950.765,E2 26950.765} C_VEL
LIN {X 0,Y 577.294,Z 189.418,A -85,B 0,C 180,E1 26947.856,E2 26947.856} C_VEL
LIN {X 0,Y 583.213,Z 208.044,A -85,B 0,C 180,E1 26945.409,E2 26945.409} C_VEL
LIN {X 0,Y 587.676,Z 222.923,A -85,B 0,C 180,E1 26943.607,E2 26943.607} C_VEL
LIN {X 0,Y 591.497,Z 231.262,A -85,B 0,C 180,E1 26943.232,E2 26943.232} C_VEL
LIN {X 0,Y 597.77,Z 260.926,A -85,B 0,C 180,E1 26942.428,E2 26942.428} C_VEL
LIN {X 0,Y 593.448,Z 521.748,A -85,B 0,C 180,E1 26939.075,E2 26939.075} C_VEL
LIN {X 0,Y 592.8,Z 539.8,A -85,B 0,C 180,E1 26938.756,E2 26938.756} C_VEL
LIN {X 0,Y 591.962,Z 557.109,A -85,B 0,C 180,E1 26938.34,E2 26938.34} C_VEL
LIN {X 0,Y 590.959,Z 574.438,A -85,B 0,C 180,E1 26937.807,E2 26937.807} C_VEL
LIN {X 0,Y 589.747,Z 592.326,A -85,B 0,C 180,E1 26937.13,E2 26937.13} C_VEL
LIN {X 0,Y 588.087,Z 613.959,A -85,B 0,C 180,E1 26936.123,E2 26936.123} C_VEL
LIN {X 0,Y 586.537,Z 631.713,A -85,B 0,C 180,E1 26935.114,E2 26935.114} C_VEL
LIN {X 0,Y 585.136,Z 647.085,A -85,B 0,C 180,E1 26934.101,E2 26934.101} C_VEL
LIN {X 0,Y 583.806,Z 661.261,A -85,B 0,C 180,E1 26933.035,E2 26933.035} C_VEL
LIN {X 0,Y 582.494,Z 674.973,A -85,B 0,C 180,E1 26931.866,E2 26931.866} C_VEL
LIN {X 0,Y 581.236,Z 688.148,A -85,B 0,C 180,E1 26930.594,E2 26930.594} C_VEL
LIN {X 0,Y 580.035,Z 701.335,A -85,B 0,C 180,E1 26929.148,E2 26929.148} C_VEL
LIN {X 0,Y 578.705,Z 716.741,A -85,B 0,C 180,E1 26927.182,E2 26927.182} C_VEL
LIN {X 0,Y 577.849,Z 727.582,A -85,B 0,C 180,E1 26925.555,E2 26925.555} C_VEL
LIN {X 0,Y 577.196,Z 736.994,A -85,B 0,C 180,E1 26923.931,E2 26923.931} C_VEL
LIN {X 0,Y 576.711,Z 745.114,A -85,B 0,C 180,E1 26922.311,E2 26922.311} C_VEL
LIN {X 0,Y 576.38,Z 752.05,A -85,B 0,C 180,E1 26920.696,E2 26920.696} C_VEL
LIN {X 0,Y 576.153,Z 757.92,A -85,B 0,C 180,E1 26919.075,E2 26919.075} C_VEL
LIN {X 0,Y 576.017,Z 762.958,A -85,B 0,C 180,E1 26917.379,E2 26917.379} C_VEL
LIN {X 0,Y 575.949,Z 766.923,A -85,B 0,C 180,E1 26915.678,E2 26915.678} C_VEL
LIN {X 0,Y 575.923,Z 770.12,A -85,B 0,C 180,E1 26913.782,E2 26913.782} C_VEL
LIN {X 0,Y 575.908,Z 772.318,A -85,B 0,C 180,E1 26911.393,E2 26911.393} C_VEL
LIN {X 0,Y 575.91,Z 772.582,A -85,B 0,C 180,E1 26909.503,E2 26909.503} C_VEL
LIN {X 0,Y 575.916,Z 771.696,A -85,B 0,C 180,E1 26907.712,E2 26907.712} C_VEL
LIN {X 0,Y 575.926,Z 769.826,A -85,B 0,C 180,E1 26906.018,E2 26906.018} C_VEL
LIN {X 0,Y 575.949,Z 766.923,A -85,B 0,C 180,E1 26904.322,E2 26904.322} C_VEL
LIN {X 0,Y 576.019,Z 762.958,A -85,B 0,C 180,E1 26902.621,E2 26902.621} C_VEL
LIN {X 0,Y 576.153,Z 757.886,A -85,B 0,C 180,E1 26900.915,E2 26900.915} C_VEL
LIN {X 0,Y 576.38,Z 752.05,A -85,B 0,C 180,E1 26899.304,E2 26899.304} C_VEL
LIN {X 0,Y 576.712,Z 745.114,A -85,B 0,C 180,E1 26897.689,E2 26897.689} C_VEL
LIN {X 0,Y 577.196,Z 736.994,A -85,B 0,C 180,E1 26896.069,E2 26896.069} C_VEL
LIN {X 0,Y 577.898,Z 726.963,A -85,B 0,C 180,E1 26894.343,E2 26894.343} C_VEL
LIN {X 0,Y 579.013,Z 713.009,A -85,B 0,C 180,E1 26892.309,E2 26892.309} C_VEL
LIN {X 0,Y 580.086,Z 700.719,A -85,B 0,C 180,E1 26890.781,E2 26890.781} C_VEL
LIN {X 0,Y 581.236,Z 688.148,A -85,B 0,C 180,E1 26889.406,E2 26889.406} C_VEL
LIN {X 0,Y 582.494,Z 674.972,A -85,B 0,C 180,E1 26888.134,E2 26888.134} C_VEL
LIN {X 0,Y 583.806,Z 661.261,A -85,B 0,C 180,E1 26886.965,E2 26886.965} C_VEL
LIN {X 0,Y 585.217,Z 646.226,A -85,B 0,C 180,E1 26885.837,E2 26885.837} C_VEL
LIN {X 0,Y 587.01,Z 626.841,A -85,B 0,C 180,E1 26884.584,E2 26884.584} C_VEL
LIN {X 0,Y 588.625,Z 607.057,A -85,B 0,C 180,E1 26883.536,E2 26883.536} C_VEL
LIN {X 0,Y 589.828,Z 591.08,A -85,B 0,C 180,E1 26882.819,E2 26882.819} C_VEL
LIN {X 0,Y 590.955,Z 574.511,A -85,B 0,C 180,E1 26882.195,E2 26882.195} C_VEL
LIN {X 0,Y 591.963,Z 557.107,A -85,B 0,C 180,E1 26881.66,E2 26881.66} C_VEL
LIN {X 0,Y 592.799,Z 539.803,A -85,B 0,C 180,E1 26881.244,E2 26881.244} C_VEL
LIN {X 0,Y 593.443,Z 521.89,A -85,B 0,C 180,E1 26880.928,E2 26880.928} C_VEL
LIN {X 0,Y 597.76,Z 261.56,A -85,B 0,C 180,E1 26877.58,E2 26877.58} C_VEL
LIN {X 0,Y 597.127,Z 256.974,A -85,B 0,C 180,E1 26877.478,E2 26877.478} C_VEL
LIN {X 0,Y 590.93,Z 229.585,A -85,B 0,C 180,E1 26876.708,E2 26876.708} C_VEL
LIN {X 0,Y 587.675,Z 222.92,A -85,B 0,C 180,E1 26876.393,E2 26876.393} C_VEL
LIN {X 0,Y 582.492,Z 205.652,A -85,B 0,C 180,E1 26874.286,E2 26874.286} C_VEL
LIN {X 0,Y 577.287,Z 189.393,A -85,B 0,C 180,E1 26872.135,E2 26872.135} C_VEL
LIN {X 0,Y 577.232,Z 189.268,A -85,B 0,C 180,E1 26869.199,E2 26869.199} C_VEL
LIN {X 0,Y 577.235,Z 189.263,A -85,B 0,C 180,E1 26865.819,E2 26865.819} C_VEL
LIN {X 0,Y 577.273,Z 189.257,A -85,B 0,C 180,E1 26862.751,E2 26862.751} C_VEL
LIN {X 0,Y 577.222,Z 189.246,A -85,B 0,C 180,E1 26859.579,E2 26859.579} C_VEL
LIN {X 0,Y 577.284,Z 189.248,A -85,B 0,C 180,E1 26856.448,E2 26856.448} C_VEL
LIN {X 0,Y 577.231,Z 189.255,A -85,B 0,C 180,E1 26853.306,E2 26853.306} C_VEL
LIN {X 0,Y 577.228,Z 189.243,A -85,B 0,C 180,E1 26849.926,E2 26849.926} C_VEL
LIN {X 0,Y 577.278,Z 189.226,A -85,B 0,C 180,E1 26846.877,E2 26846.877} C_VEL
LIN {X 0,Y 577.224,Z 189.262,A -85,B 0,C 180,E1 26843.696,E2 26843.696} C_VEL
LIN {X 0,Y 577.281,Z 189.259,A -85,B 0,C 180,E1 26840.586,E2 26840.586} C_VEL
LIN {X 0,Y 577.229,Z 189.248,A -85,B 0,C 180,E1 26837.542,E2 26837.542} C_VEL
LIN {X 0,Y 577.236,Z 189.255,A -85,B 0,C 180,E1 26834.239,E2 26834.239} C_VEL
LIN {X 0,Y 577.262,Z 189.256,A -85,B 0,C 180,E1 26831.186,E2 26831.186} C_VEL
LIN {X 0,Y 577.224,Z 189.247,A -85,B 0,C 180,E1 26828.066,E2 26828.066} C_VEL
LIN {X 0,Y 577.292,Z 189.26,A -85,B 0,C 180,E1 26824.968,E2 26824.968} C_VEL
LIN {X 0,Y 577.225,Z 189.256,A -85,B 0,C 180,E1 26821.787,E2 26821.787} C_VEL
LIN {X 0,Y 577.243,Z 189.249,A -85,B 0,C 180,E1 26818.511,E2 26818.511} C_VEL
LIN {X 0,Y 577.254,Z 189.261,A -85,B 0,C 180,E1 26815.43,E2 26815.43} C_VEL
LIN {X 0,Y 577.225,Z 189.254,A -85,B 0,C 180,E1 26812.235,E2 26812.235} C_VEL
LIN {X 0,Y 577.289,Z 189.253,A -85,B 0,C 180,E1 26809.092,E2 26809.092} C_VEL
LIN {X 0,Y 577.224,Z 189.261,A -85,B 0,C 180,E1 26805.965,E2 26805.965} C_VEL
LIN {X 0,Y 577.251,Z 189.253,A -85,B 0,C 180,E1 26802.771,E2 26802.771} C_VEL
LIN {X 0,Y 577.245,Z 189.262,A -85,B 0,C 180,E1 26799.73,E2 26799.73} C_VEL
LIN {X 0,Y 577.23,Z 189.263,A -85,B 0,C 180,E1 26796.521,E2 26796.521} C_VEL
LIN {X 0,Y 577.276,Z 189.222,A -85,B 0,C 180,E1 26793.456,E2 26793.456} C_VEL
LIN {X 0,Y 577.222,Z 189.251,A -85,B 0,C 180,E1 26790.302,E2 26790.302} C_VEL
LIN {X 0,Y 577.275,Z 189.25,A -85,B 0,C 180,E1 26787.17,E2 26787.17} C_VEL
LIN {X 0,Y 577.228,Z 189.232,A -85,B 0,C 180,E1 26784.039,E2 26784.039} C_VEL
LIN {X 0,Y 577.231,Z 189.264,A -85,B 0,C 180,E1 26780.732,E2 26780.732} C_VEL
LIN {X 0,Y 577.274,Z 189.264,A -85,B 0,C 180,E1 26777.689,E2 26777.689} C_VEL
LIN {X 0,Y 577.223,Z 189.265,A -85,B 0,C 180,E1 26774.544,E2 26774.544} C_VEL
LIN {X 0,Y 577.287,Z 189.261,A -85,B 0,C 180,E1 26771.411,E2 26771.411} C_VEL
LIN {X 0,Y 577.223,Z 189.266,A -85,B 0,C 180,E1 26768.447,E2 26768.447} C_VEL
LIN {X 0,Y 577.255,Z 189.263,A -85,B 0,C 180,E1 26765.221,E2 26765.221} C_VEL
LIN {X 0,Y 577.237,Z 189.265,A -85,B 0,C 180,E1 26762.238,E2 26762.238} C_VEL
LIN {X 0,Y 577.228,Z 189.267,A -85,B 0,C 180,E1 26758.896,E2 26758.896} C_VEL
LIN {X 0,Y 577.291,Z 189.261,A -85,B 0,C 180,E1 26755.754,E2 26755.754} C_VEL
LIN {X 0,Y 577.226,Z 189.265,A -85,B 0,C 180,E1 26752.589,E2 26752.589} C_VEL
LIN {X 0,Y 577.258,Z 189.264,A -85,B 0,C 180,E1 26749.422,E2 26749.422} C_VEL
LIN {X 0,Y 577.264,Z 189.262,A -85,B 0,C 180,E1 26748.105,E2 26748.105} C_VEL
LIN {X 0,Y 576.32,Z 189.383,A -85,B 0,C 180,E1 26747.34,E2 26747.34} C_VEL
LIN {X 0,Y 569.821,Z 190.194,A -85,B 0,C 180,E1 26745.194,E2 26745.194} C_VEL
LIN {X 0,Y 569.288,Z 190.256,A -85,B 0,C 180,E1 26744.635,E2 26744.635} C_VEL
LIN {X 0,Y 569.302,Z 190.253,A -85,B 0,C 180,E1 26741.343,E2 26741.343} C_VEL
LIN {X 0,Y 569.317,Z 190.253,A -85,B 0,C 180,E1 26738.279,E2 26738.279} C_VEL
LIN {X 0,Y 569.287,Z 190.256,A -85,B 0,C 180,E1 26735.139,E2 26735.139} C_VEL
LIN {X 0,Y 569.35,Z 190.247,A -85,B 0,C 180,E1 26732.013,E2 26732.013} C_VEL
LIN {X 0,Y 569.283,Z 190.256,A -85,B 0,C 180,E1 26728.994,E2 26728.994} C_VEL
LIN {X 0,Y 569.327,Z 190.252,A -85,B 0,C 180,E1 26725.77,E2 26725.77} C_VEL
LIN {X 0,Y 569.295,Z 190.254,A -85,B 0,C 180,E1 26722.736,E2 26722.736} C_VEL
LIN {X 0,Y 569.29,Z 190.257,A -85,B 0,C 180,E1 26719.374,E2 26719.374} C_VEL
LIN {X 0,Y 569.359,Z 190.248,A -85,B 0,C 180,E1 26716.184,E2 26716.184} C_VEL
LIN {X 0,Y 569.286,Z 190.254,A -85,B 0,C 180,E1 26713.051,E2 26713.051} C_VEL
LIN {X 0,Y 569.308,Z 190.256,A -85,B 0,C 180,E1 26709.76,E2 26709.76} C_VEL
LIN {X 0,Y 569.299,Z 190.256,A -85,B 0,C 180,E1 26706.836,E2 26706.836} C_VEL
LIN {X 0,Y 569.288,Z 190.253,A -85,B 0,C 180,E1 26703.509,E2 26703.509} C_VEL
LIN {X 0,Y 569.358,Z 190.247,A -85,B 0,C 180,E1 26700.378,E2 26700.378} C_VEL
LIN {X 0,Y 569.286,Z 190.255,A -85,B 0,C 180,E1 26697.255,E2 26697.255} C_VEL
LIN {X 0,Y 569.312,Z 190.252,A -85,B 0,C 180,E1 26693.965,E2 26693.965} C_VEL
LIN {X 0,Y 569.307,Z 190.254,A -85,B 0,C 180,E1 26690.918,E2 26690.918} C_VEL
LIN {X 0,Y 569.289,Z 190.254,A -85,B 0,C 180,E1 26687.684,E2 26687.684} C_VEL
LIN {X 0,Y 569.352,Z 190.25,A -85,B 0,C 180,E1 26684.485,E2 26684.485} C_VEL
LIN {X 0,Y 569.29,Z 190.253,A -85,B 0,C 180,E1 26681.331,E2 26681.331} C_VEL
LIN {X 0,Y 569.303,Z 190.251,A -85,B 0,C 180,E1 26678.059,E2 26678.059} C_VEL
LIN {X 0,Y 569.316,Z 190.209,A -85,B 0,C 180,E1 26674.929,E2 26674.929} C_VEL
LIN {X 0,Y 569.286,Z 190.253,A -85,B 0,C 180,E1 26671.791,E2 26671.791} C_VEL
LIN {X 0,Y 569.353,Z 190.198,A -85,B 0,C 180,E1 26668.649,E2 26668.649} C_VEL
LIN {X 0,Y 569.289,Z 190.239,A -85,B 0,C 180,E1 26665.488,E2 26665.488} C_VEL
LIN {X 0,Y 569.298,Z 190.241,A -85,B 0,C 180,E1 26662.186,E2 26662.186} C_VEL
LIN {X 0,Y 569.323,Z 190.251,A -85,B 0,C 180,E1 26659.135,E2 26659.135} C_VEL
LIN {X 0,Y 569.284,Z 190.246,A -85,B 0,C 180,E1 26655.902,E2 26655.902} C_VEL
LIN {X 0,Y 569.349,Z 190.234,A -85,B 0,C 180,E1 26652.784,E2 26652.784} C_VEL
LIN {X 0,Y 569.292,Z 190.251,A -85,B 0,C 180,E1 26649.605,E2 26649.605} C_VEL
LIN {X 0,Y 569.291,Z 190.248,A -85,B 0,C 180,E1 26646.252,E2 26646.252} C_VEL
LIN {X 0,Y 569.34,Z 190.239,A -85,B 0,C 180,E1 26643.121,E2 26643.121} C_VEL
LIN {X 0,Y 569.284,Z 190.251,A -85,B 0,C 180,E1 26640,E2 26640} C_VEL
LIN {X 0,Y 569.339,Z 190.234,A -85,B 0,C 180,E1 26636.879,E2 26636.879} C_VEL
LIN {X 0,Y 569.294,Z 190.249,A -85,B 0,C 180,E1 26633.748,E2 26633.748} C_VEL
LIN {X 0,Y 569.292,Z 190.249,A -85,B 0,C 180,E1 26630.395,E2 26630.395} C_VEL
LIN {X 0,Y 569.35,Z 190.234,A -85,B 0,C 180,E1 26627.216,E2 26627.216} C_VEL
LIN {X 0,Y 569.286,Z 190.251,A -85,B 0,C 180,E1 26624.098,E2 26624.098} C_VEL
LIN {X 0,Y 569.32,Z 190.252,A -85,B 0,C 180,E1 26620.866,E2 26620.866} C_VEL
LIN {X 0,Y 569.301,Z 190.24,A -85,B 0,C 180,E1 26617.814,E2 26617.814} C_VEL
LIN {X 0,Y 569.29,Z 190.245,A -85,B 0,C 180,E1 26614.509,E2 26614.509} C_VEL
LIN {X 0,Y 569.355,Z 190.198,A -85,B 0,C 180,E1 26611.351,E2 26611.351} C_VEL
LIN {X 0,Y 569.29,Z 190.252,A -85,B 0,C 180,E1 26608.203,E2 26608.203} C_VEL
LIN {X 0,Y 569.305,Z 190.225,A -85,B 0,C 180,E1 26604.919,E2 26604.919} C_VEL
LIN {X 0,Y 569.318,Z 190.252,A -85,B 0,C 180,E1 26601.814,E2 26601.814} C_VEL
LIN {X 0,Y 569.288,Z 190.251,A -85,B 0,C 180,E1 26598.579,E2 26598.579} C_VEL
LIN {X 0,Y 569.344,Z 190.23,A -85,B 0,C 180,E1 26595.373,E2 26595.373} C_VEL
LIN {X 0,Y 569.29,Z 190.238,A -85,B 0,C 180,E1 26592.268,E2 26592.268} C_VEL
LIN {X 0,Y 569.288,Z 190.202,A -85,B 0,C 180,E1 26588.915,E2 26588.915} C_VEL
LIN {X 0,Y 569.343,Z 190.583,A -85,B 0,C 180,E1 26588.299,E2 26588.299} C_VEL
LIN {X 0,Y 575.664,Z 210.099,A -85,B 0,C 180,E1 26585.699,E2 26585.699} C_VEL
LIN {X 0,Y 579.401,Z 222.507,A -85,B 0,C 180,E1 26584.158,E2 26584.158} C_VEL
LIN {X 0,Y 585.119,Z 234.405,A -85,B 0,C 180,E1 26583.595,E2 26583.595} C_VEL
LIN {X 0,Y 590.987,Z 262.286,A -85,B 0,C 180,E1 26582.825,E2 26582.825} C_VEL
LIN {X 0,Y 586.445,Z 521.795,A -85,B 0,C 180,E1 26579.452,E2 26579.452} C_VEL
LIN {X 0,Y 585.772,Z 539.746,A -85,B 0,C 180,E1 26579.131,E2 26579.131} C_VEL
LIN {X 0,Y 584.889,Z 557.091,A -85,B 0,C 180,E1 26578.709,E2 26578.709} C_VEL
LIN {X 0,Y 583.844,Z 574.261,A -85,B 0,C 180,E1 26578.176,E2 26578.176} C_VEL
LIN {X 0,Y 582.567,Z 592.149,A -85,B 0,C 180,E1 26577.493,E2 26577.493} C_VEL
LIN {X 0,Y 580.809,Z 613.968,A -85,B 0,C 180,E1 26576.465,E2 26576.465} C_VEL
LIN {X 0,Y 579.192,Z 631.535,A -85,B 0,C 180,E1 26575.455,E2 26575.455} C_VEL
LIN {X 0,Y 577.711,Z 646.907,A -85,B 0,C 180,E1 26574.431,E2 26574.431} C_VEL
LIN {X 0,Y 576.308,Z 661.083,A -85,B 0,C 180,E1 26573.353,E2 26573.353} C_VEL
LIN {X 0,Y 574.924,Z 674.794,A -85,B 0,C 180,E1 26572.169,E2 26572.169} C_VEL
LIN {X 0,Y 573.585,Z 688.057,A -85,B 0,C 180,E1 26570.872,E2 26570.872} C_VEL
LIN {X 0,Y 572.287,Z 701.431,A -85,B 0,C 180,E1 26569.385,E2 26569.385} C_VEL
LIN {X 0,Y 570.832,Z 717.264,A -85,B 0,C 180,E1 26567.322,E2 26567.322} C_VEL
LIN {X 0,Y 569.935,Z 728.022,A -85,B 0,C 180,E1 26565.673,E2 26565.673} C_VEL
LIN {X 0,Y 569.285,Z 736.815,A -85,B 0,C 180,E1 26564.129,E2 26564.129} C_VEL
LIN {X 0,Y 568.767,Z 744.936,A -85,B 0,C 180,E1 26562.486,E2 26562.486} C_VEL
LIN {X 0,Y 568.412,Z 751.873,A -85,B 0,C 180,E1 26560.848,E2 26560.848} C_VEL
LIN {X 0,Y 568.164,Z 757.934,A -85,B 0,C 180,E1 26559.145,E2 26559.145} C_VEL
LIN {X 0,Y 568.018,Z 763.051,A -85,B 0,C 180,E1 26557.382,E2 26557.382} C_VEL
LIN {X 0,Y 567.936,Z 767.578,A -85,B 0,C 180,E1 26555.353,E2 26555.353} C_VEL
LIN {X 0,Y 567.911,Z 770.904,A -85,B 0,C 180,E1 26553.027,E2 26553.027} C_VEL
LIN {X 0,Y 567.913,Z 772.232,A -85,B 0,C 180,E1 26551.11,E2 26551.11} C_VEL
LIN {X 0,Y 567.913,Z 772.378,A -85,B 0,C 180,E1 26549.395,E2 26549.395} C_VEL
LIN {X 0,Y 567.917,Z 771.433,A -85,B 0,C 180,E1 26547.579,E2 26547.579} C_VEL
LIN {X 0,Y 567.927,Z 769.503,A -85,B 0,C 180,E1 26545.861,E2 26545.861} C_VEL
LIN {X 0,Y 567.956,Z 766.444,A -85,B 0,C 180,E1 26544.094,E2 26544.094} C_VEL
LIN {X 0,Y 568.027,Z 762.512,A -85,B 0,C 180,E1 26542.415,E2 26542.415} C_VEL
LIN {X 0,Y 568.172,Z 757.709,A -85,B 0,C 180,E1 26540.786,E2 26540.786} C_VEL
LIN {X 0,Y 568.412,Z 751.873,A -85,B 0,C 180,E1 26539.152,E2 26539.152} C_VEL
LIN {X 0,Y 568.768,Z 744.936,A -85,B 0,C 180,E1 26537.514,E2 26537.514} C_VEL
LIN {X 0,Y 569.285,Z 736.815,A -85,B 0,C 180,E1 26535.871,E2 26535.871} C_VEL
LIN {X 0,Y 570.037,Z 726.784,A -85,B 0,C 180,E1 26534.121,E2 26534.121} C_VEL
LIN {X 0,Y 571.229,Z 712.831,A -85,B 0,C 180,E1 26532.059,E2 26532.059} C_VEL
LIN {X 0,Y 572.365,Z 700.54,A -85,B 0,C 180,E1 26530.511,E2 26530.511} C_VEL
LIN {X 0,Y 573.587,Z 688.051,A -85,B 0,C 180,E1 26529.127,E2 26529.127} C_VEL
LIN {X 0,Y 574.924,Z 674.794,A -85,B 0,C 180,E1 26527.83,E2 26527.83} C_VEL
LIN {X 0,Y 576.308,Z 661.082,A -85,B 0,C 180,E1 26526.647,E2 26526.647} C_VEL
LIN {X 0,Y 577.776,Z 646.267,A -85,B 0,C 180,E1 26525.523,E2 26525.523} C_VEL
LIN {X 0,Y 579.607,Z 627.503,A -85,B 0,C 180,E1 26524.291,E2 26524.291} C_VEL
LIN {X 0,Y 581.338,Z 607.527,A -85,B 0,C 180,E1 26523.211,E2 26523.211} C_VEL
LIN {X 0,Y 582.654,Z 590.904,A -85,B 0,C 180,E1 26522.456,E2 26522.456} C_VEL
LIN {X 0,Y 583.845,Z 574.26,A -85,B 0,C 180,E1 26521.824,E2 26521.824} C_VEL
LIN {X 0,Y 584.901,Z 556.894,A -85,B 0,C 180,E1 26521.285,E2 26521.285} C_VEL
LIN {X 0,Y 585.779,Z 539.593,A -85,B 0,C 180,E1 26520.866,E2 26520.866} C_VEL
LIN {X 0,Y 586.452,Z 521.588,A -85,B 0,C 180,E1 26520.545,E2 26520.545} C_VEL
LIN {X 0,Y 590.997,Z 261.594,A -85,B 0,C 180,E1 26517.166,E2 26517.166} C_VEL
LIN {X 0,Y 584.631,Z 233.053,A -85,B 0,C 180,E1 26516.354,E2 26516.354} C_VEL
LIN {X 0,Y 579.279,Z 222.161,A -85,B 0,C 180,E1 26515.816,E2 26515.816} C_VEL
LIN {X 0,Y 572.886,Z 201.299,A -85,B 0,C 180,E1 26513.154,E2 26513.154} C_VEL
LIN {X 0,Y 569.307,Z 190.373,A -85,B 0,C 180,E1 26511.648,E2 26511.648} C_VEL
LIN {X 0,Y 569.335,Z 190.239,A -85,B 0,C 180,E1 26508.681,E2 26508.681} C_VEL
LIN {X 0,Y 569.286,Z 190.251,A -85,B 0,C 180,E1 26505.488,E2 26505.488} C_VEL
LIN {X 0,Y 569.333,Z 190.252,A -85,B 0,C 180,E1 26502.272,E2 26502.272} C_VEL
LIN {X 0,Y 569.295,Z 190.237,A -85,B 0,C 180,E1 26499.22,E2 26499.22} C_VEL
LIN {X 0,Y 569.293,Z 190.236,A -85,B 0,C 180,E1 26495.918,E2 26495.918} C_VEL
LIN {X 0,Y 569.347,Z 190.244,A -85,B 0,C 180,E1 26492.743,E2 26492.743} C_VEL
LIN {X 0,Y 569.283,Z 190.225,A -85,B 0,C 180,E1 26489.623,E2 26489.623} C_VEL
LIN {X 0,Y 569.336,Z 190.222,A -85,B 0,C 180,E1 26486.493,E2 26486.493} C_VEL
LIN {X 0,Y 569.297,Z 190.251,A -85,B 0,C 180,E1 26483.387,E2 26483.387} C_VEL
LIN {X 0,Y 569.29,Z 190.251,A -85,B 0,C 180,E1 26480.027,E2 26480.027} C_VEL
LIN {X 0,Y 569.352,Z 190.234,A -85,B 0,C 180,E1 26476.844,E2 26476.844} C_VEL
LIN {X 0,Y 569.284,Z 190.244,A -85,B 0,C 180,E1 26473.795,E2 26473.795} C_VEL
LIN {X 0,Y 569.331,Z 190.249,A -85,B 0,C 180,E1 26470.627,E2 26470.627} C_VEL
LIN {X 0,Y 569.291,Z 190.235,A -85,B 0,C 180,E1 26467.57,E2 26467.57} C_VEL
LIN {X 0,Y 569.291,Z 190.245,A -85,B 0,C 180,E1 26464.23,E2 26464.23} C_VEL
LIN {X 0,Y 569.357,Z 190.245,A -85,B 0,C 180,E1 26461.006,E2 26461.006} C_VEL
LIN {X 0,Y 569.283,Z 190.237,A -85,B 0,C 180,E1 26457.886,E2 26457.886} C_VEL
LIN {X 0,Y 569.314,Z 190.248,A -85,B 0,C 180,E1 26454.659,E2 26454.659} C_VEL
LIN {X 0,Y 569.294,Z 190.243,A -85,B 0,C 180,E1 26451.719,E2 26451.719} C_VEL
LIN {X 0,Y 569.292,Z 190.239,A -85,B 0,C 180,E1 26448.45,E2 26448.45} C_VEL
LIN {X 0,Y 569.337,Z 190.25,A -85,B 0,C 180,E1 26445.351,E2 26445.351} C_VEL
LIN {X 0,Y 569.286,Z 190.246,A -85,B 0,C 180,E1 26442.145,E2 26442.145} C_VEL
LIN {X 0,Y 569.333,Z 190.237,A -85,B 0,C 180,E1 26439.006,E2 26439.006} C_VEL
LIN {X 0,Y 569.292,Z 190.252,A -85,B 0,C 180,E1 26435.953,E2 26435.953} C_VEL
LIN {X 0,Y 569.287,Z 190.201,A -85,B 0,C 180,E1 26432.602,E2 26432.602} C_VEL
LIN {X 0,Y 569.342,Z 190.24,A -85,B 0,C 180,E1 26429.499,E2 26429.499} C_VEL
LIN {X 0,Y 569.283,Z 190.237,A -85,B 0,C 180,E1 26426.348,E2 26426.348} C_VEL
LIN {X 0,Y 569.333,Z 190.229,A -85,B 0,C 180,E1 26423.201,E2 26423.201} C_VEL
LIN {X 0,Y 569.287,Z 190.253,A -85,B 0,C 180,E1 26420.258,E2 26420.258} C_VEL
LIN {X 0,Y 569.313,Z 190.253,A -85,B 0,C 180,E1 26417.043,E2 26417.043} C_VEL
LIN {X 0,Y 569.314,Z 190.254,A -85,B 0,C 180,E1 26413.919,E2 26413.919} C_VEL
LIN {X 0,Y 569.292,Z 190.252,A -85,B 0,C 180,E1 26410.789,E2 26410.789} C_VEL
LIN {X 0,Y 569.349,Z 190.248,A -85,B 0,C 180,E1 26407.667,E2 26407.667} C_VEL
LIN {X 0,Y 569.287,Z 190.255,A -85,B 0,C 180,E1 26404.436,E2 26404.436} C_VEL
LIN {X 0,Y 569.311,Z 190.252,A -85,B 0,C 180,E1 26401.201,E2 26401.201} C_VEL
LIN {X 0,Y 569.296,Z 190.255,A -85,B 0,C 180,E1 26398.304,E2 26398.304} C_VEL
LIN {X 0,Y 569.292,Z 190.255,A -85,B 0,C 180,E1 26395.002,E2 26395.002} C_VEL
LIN {X 0,Y 569.351,Z 190.25,A -85,B 0,C 180,E1 26391.855,E2 26391.855} C_VEL
LIN {X 0,Y 569.286,Z 190.257,A -85,B 0,C 180,E1 26388.746,E2 26388.746} C_VEL
LIN {X 0,Y 569.33,Z 190.25,A -85,B 0,C 180,E1 26385.585,E2 26385.585} C_VEL
LIN {X 0,Y 569.288,Z 190.256,A -85,B 0,C 180,E1 26384.635,E2 26384.635} C_VEL
LIN {X 0,Y 568.317,Z 190.378,A -85,B 0,C 180,E1 26383.86,E2 26383.86} C_VEL
LIN {X 0,Y 561.802,Z 191.189,A -85,B 0,C 180,E1 26381.627,E2 26381.627} C_VEL
LIN {X 0,Y 561.35,Z 191.245,A -85,B 0,C 180,E1 26381.116,E2 26381.116} C_VEL
LIN {X 0,Y 561.421,Z 191.236,A -85,B 0,C 180,E1 26377.881,E2 26377.881} C_VEL
LIN {X 0,Y 561.349,Z 191.243,A -85,B 0,C 180,E1 26374.699,E2 26374.699} C_VEL
LIN {X 0,Y 561.354,Z 191.247,A -85,B 0,C 180,E1 26371.327,E2 26371.327} C_VEL
LIN {X 0,Y 561.378,Z 191.242,A -85,B 0,C 180,E1 26368.367,E2 26368.367} C_VEL
LIN {X 0,Y 561.345,Z 191.244,A -85,B 0,C 180,E1 26365.096,E2 26365.096} C_VEL
LIN {X 0,Y 561.401,Z 191.241,A -85,B 0,C 180,E1 26361.913,E2 26361.913} C_VEL
LIN {X 0,Y 561.354,Z 191.244,A -85,B 0,C 180,E1 26358.806,E2 26358.806} C_VEL
LIN {X 0,Y 561.352,Z 191.244,A -85,B 0,C 180,E1 26355.456,E2 26355.456} C_VEL
LIN {X 0,Y 561.41,Z 191.24,A -85,B 0,C 180,E1 26352.271,E2 26352.271} C_VEL
LIN {X 0,Y 561.347,Z 191.244,A -85,B 0,C 180,E1 26349.133,E2 26349.133} C_VEL
LIN {X 0,Y 561.383,Z 191.241,A -85,B 0,C 180,E1 26345.932,E2 26345.932} C_VEL
LIN {X 0,Y 561.372,Z 191.243,A -85,B 0,C 180,E1 26342.762,E2 26342.762} C_VEL
LIN {X 0,Y 561.347,Z 191.243,A -85,B 0,C 180,E1 26339.497,E2 26339.497} C_VEL
LIN {X 0,Y 561.415,Z 191.236,A -85,B 0,C 180,E1 26336.371,E2 26336.371} C_VEL
LIN {X 0,Y 561.349,Z 191.242,A -85,B 0,C 180,E1 26333.244,E2 26333.244} C_VEL
LIN {X 0,Y 561.371,Z 191.242,A -85,B 0,C 180,E1 26329.987,E2 26329.987} C_VEL
LIN {X 0,Y 561.373,Z 191.243,A -85,B 0,C 180,E1 26326.909,E2 26326.909} C_VEL
LIN {X 0,Y 561.349,Z 191.243,A -85,B 0,C 180,E1 26323.691,E2 26323.691} C_VEL
LIN {X 0,Y 561.42,Z 191.238,A -85,B 0,C 180,E1 26320.502,E2 26320.502} C_VEL
LIN {X 0,Y 561.348,Z 191.24,A -85,B 0,C 180,E1 26317.402,E2 26317.402} C_VEL
LIN {X 0,Y 561.355,Z 191.212,A -85,B 0,C 180,E1 26314.008,E2 26314.008} C_VEL
LIN {X 0,Y 561.399,Z 191.236,A -85,B 0,C 180,E1 26310.86,E2 26310.86} C_VEL
LIN {X 0,Y 561.341,Z 191.185,A -85,B 0,C 180,E1 26307.704,E2 26307.704} C_VEL
LIN {X 0,Y 561.394,Z 191.238,A -85,B 0,C 180,E1 26304.493,E2 26304.493} C_VEL
LIN {X 0,Y 561.354,Z 191.228,A -85,B 0,C 180,E1 26301.417,E2 26301.417} C_VEL
LIN {X 0,Y 561.351,Z 191.234,A -85,B 0,C 180,E1 26298.055,E2 26298.055} C_VEL
LIN {X 0,Y 561.422,Z 191.236,A -85,B 0,C 180,E1 26294.86,E2 26294.86} C_VEL
LIN {X 0,Y 561.35,Z 191.227,A -85,B 0,C 180,E1 26291.612,E2 26291.612} C_VEL
LIN {X 0,Y 561.35,Z 191.23,A -85,B 0,C 180,E1 26288.192,E2 26288.192} C_VEL
LIN {X 0,Y 561.402,Z 191.237,A -85,B 0,C 180,E1 26285.109,E2 26285.109} C_VEL
LIN {X 0,Y 561.343,Z 191.225,A -85,B 0,C 180,E1 26281.939,E2 26281.939} C_VEL
LIN {X 0,Y 561.393,Z 191.233,A -85,B 0,C 180,E1 26278.775,E2 26278.775} C_VEL
LIN {X 0,Y 561.362,Z 191.232,A -85,B 0,C 180,E1 26275.607,E2 26275.607} C_VEL
LIN {X 0,Y 561.349,Z 191.222,A -85,B 0,C 180,E1 26272.323,E2 26272.323} C_VEL
LIN {X 0,Y 561.411,Z 191.235,A -85,B 0,C 180,E1 26269.118,E2 26269.118} C_VEL
LIN {X 0,Y 561.35,Z 191.235,A -85,B 0,C 180,E1 26265.981,E2 26265.981} C_VEL
LIN {X 0,Y 561.365,Z 191.225,A -85,B 0,C 180,E1 26262.665,E2 26262.665} C_VEL
LIN {X 0,Y 561.391,Z 191.241,A -85,B 0,C 180,E1 26259.509,E2 26259.509} C_VEL
LIN {X 0,Y 561.348,Z 191.24,A -85,B 0,C 180,E1 26256.373,E2 26256.373} C_VEL
LIN {X 0,Y 561.402,Z 191.201,A -85,B 0,C 180,E1 26253.149,E2 26253.149} C_VEL
LIN {X 0,Y 561.35,Z 191.22,A -85,B 0,C 180,E1 26250.083,E2 26250.083} C_VEL
LIN {X 0,Y 561.357,Z 191.232,A -85,B 0,C 180,E1 26246.728,E2 26246.728} C_VEL
LIN {X 0,Y 561.411,Z 191.225,A -85,B 0,C 180,E1 26243.497,E2 26243.497} C_VEL
LIN {X 0,Y 561.345,Z 191.222,A -85,B 0,C 180,E1 26240.38,E2 26240.38} C_VEL
LIN {X 0,Y 561.381,Z 191.235,A -85,B 0,C 180,E1 26237.126,E2 26237.126} C_VEL
LIN {X 0,Y 561.373,Z 191.242,A -85,B 0,C 180,E1 26233.979,E2 26233.979} C_VEL
LIN {X 0,Y 561.35,Z 191.248,A -85,B 0,C 180,E1 26230.68,E2 26230.68} C_VEL
LIN {X 0,Y 561.374,Z 191.401,A -85,B 0,C 180,E1 26228.837,E2 26228.837} C_VEL
LIN {X 0,Y 566.843,Z 208.038,A -85,B 0,C 180,E1 26226.535,E2 26226.535} C_VEL
LIN {X 0,Y 571.185,Z 222.101,A -85,B 0,C 180,E1 26224.725,E2 26224.725} C_VEL
LIN {X 0,Y 578.843,Z 237.911,A -85,B 0,C 180,E1 26223.955,E2 26223.955} C_VEL
LIN {X 0,Y 584.227,Z 263.887,A -85,B 0,C 180,E1 26223.228,E2 26223.228} C_VEL
LIN {X 0,Y 579.464,Z 522.031,A -85,B 0,C 180,E1 26219.835,E2 26219.835} C_VEL
LIN {X 0,Y 578.77,Z 539.691,A -85,B 0,C 180,E1 26219.515,E2 26219.515} C_VEL
LIN {X 0,Y 577.853,Z 556.894,A -85,B 0,C 180,E1 26219.093,E2 26219.093} C_VEL
LIN {X 0,Y 576.756,Z 574.085,A -85,B 0,C 180,E1 26218.554,E2 26218.554} C_VEL
LIN {X 0,Y 575.414,Z 591.973,A -85,B 0,C 180,E1 26217.864,E2 26217.864} C_VEL
LIN {X 0,Y 573.591,Z 613.605,A -85,B 0,C 180,E1 26216.835,E2 26216.835} C_VEL
LIN {X 0,Y 571.813,Z 631.91,A -85,B 0,C 180,E1 26215.769,E2 26215.769} C_VEL
LIN {X 0,Y 570.258,Z 647.226,A -85,B 0,C 180,E1 26214.733,E2 26214.733} C_VEL
LIN {X 0,Y 568.761,Z 661.535,A -85,B 0,C 180,E1 26213.626,E2 26213.626} C_VEL
LIN {X 0,Y 567.326,Z 675.026,A -85,B 0,C 180,E1 26212.443,E2 26212.443} C_VEL
LIN {X 0,Y 565.914,Z 688.291,A -85,B 0,C 180,E1 26211.124,E2 26211.124} C_VEL
LIN {X 0,Y 564.487,Z 702.195,A -85,B 0,C 180,E1 26209.55,E2 26209.55} C_VEL
LIN {X 0,Y 563.031,Z 717.086,A -85,B 0,C 180,E1 26207.569,E2 26207.569} C_VEL
LIN {X 0,Y 562.076,Z 727.843,A -85,B 0,C 180,E1 26205.897,E2 26205.897} C_VEL
LIN {X 0,Y 561.372,Z 736.73,A -85,B 0,C 180,E1 26204.314,E2 26204.314} C_VEL
LIN {X 0,Y 560.829,Z 744.759,A -85,B 0,C 180,E1 26202.666,E2 26202.666} C_VEL
LIN {X 0,Y 560.446,Z 751.696,A -85,B 0,C 180,E1 26201.004,E2 26201.004} C_VEL
LIN {X 0,Y 560.19,Z 757.533,A -85,B 0,C 180,E1 26199.346,E2 26199.346} C_VEL
LIN {X 0,Y 560.028,Z 762.605,A -85,B 0,C 180,E1 26197.591,E2 26197.591} C_VEL
LIN {X 0,Y 559.95,Z 766.78,A -85,B 0,C 180,E1 26195.738,E2 26195.738} C_VEL
LIN {X 0,Y 559.915,Z 770.355,A -85,B 0,C 180,E1 26193.48,E2 26193.48} C_VEL
LIN {X 0,Y 559.914,Z 772.028,A -85,B 0,C 180,E1 26191.228,E2 26191.228} C_VEL
LIN {X 0,Y 559.915,Z 772.204,A -85,B 0,C 180,E1 26189.386,E2 26189.386} C_VEL
LIN {X 0,Y 559.918,Z 771.258,A -85,B 0,C 180,E1 26187.544,E2 26187.544} C_VEL
LIN {X 0,Y 559.928,Z 769.328,A -85,B 0,C 180,E1 26185.802,E2 26185.802} C_VEL
LIN {X 0,Y 559.959,Z 766.352,A -85,B 0,C 180,E1 26184.05,E2 26184.05} C_VEL
LIN {X 0,Y 560.032,Z 762.336,A -85,B 0,C 180,E1 26182.306,E2 26182.306} C_VEL
LIN {X 0,Y 560.2,Z 757.199,A -85,B 0,C 180,E1 26180.55,E2 26180.55} C_VEL
LIN {X 0,Y 560.482,Z 750.897,A -85,B 0,C 180,E1 26178.789,E2 26178.789} C_VEL
LIN {X 0,Y 560.956,Z 742.885,A -85,B 0,C 180,E1 26176.918,E2 26176.918} C_VEL
LIN {X 0,Y 561.83,Z 730.936,A -85,B 0,C 180,E1 26174.625,E2 26174.625} C_VEL
LIN {X 0,Y 562.711,Z 720.491,A -85,B 0,C 180,E1 26172.938,E2 26172.938} C_VEL
LIN {X 0,Y 563.674,Z 710.277,A -85,B 0,C 180,E1 26171.489,E2 26171.489} C_VEL
LIN {X 0,Y 564.835,Z 698.581,A -85,B 0,C 180,E1 26170.025,E2 26170.025} C_VEL
LIN {X 0,Y 566.183,Z 685.792,A -85,B 0,C 180,E1 26168.615,E2 26168.615} C_VEL
LIN {X 0,Y 567.669,Z 671.81,A -85,B 0,C 180,E1 26167.259,E2 26167.259} C_VEL
LIN {X 0,Y 569.68,Z 653.132,A -85,B 0,C 180,E1 26165.699,E2 26165.699} C_VEL
LIN {X 0,Y 571.39,Z 636.196,A -85,B 0,C 180,E1 26164.506,E2 26164.506} C_VEL
LIN {X 0,Y 572.933,Z 620.142,A -85,B 0,C 180,E1 26163.528,E2 26163.528} C_VEL
LIN {X 0,Y 574.333,Z 604.827,A -85,B 0,C 180,E1 26162.725,E2 26162.725} C_VEL
LIN {X 0,Y 575.703,Z 588.239,A -85,B 0,C 180,E1 26161.982,E2 26161.982} C_VEL
LIN {X 0,Y 576.915,Z 571.854,A -85,B 0,C 180,E1 26161.37,E2 26161.37} C_VEL
LIN {X 0,Y 578.016,Z 554.283,A -85,B 0,C 180,E1 26160.835,E2 26160.835} C_VEL
LIN {X 0,Y 579.087,Z 533.571,A -85,B 0,C 180,E1 26160.355,E2 26160.355} C_VEL
LIN {X 0,Y 579.873,Z 503.57,A -85,B 0,C 180,E1 26159.908,E2 26159.908} C_VEL
LIN {X 0,Y 584.192,Z 262.796,A -85,B 0,C 180,E1 26156.754,E2 26156.754} C_VEL
LIN {X 0,Y 578.367,Z 236.521,A -85,B 0,C 180,E1 26155.993,E2 26155.993} C_VEL
LIN {X 0,Y 571.068,Z 221.768,A -85,B 0,C 180,E1 26155.247,E2 26155.247} C_VEL
LIN {X 0,Y 564.854,Z 201.894,A -85,B 0,C 180,E1 26152.638,E2 26152.638} C_VEL
LIN {X 0,Y 561.368,Z 191.352,A -85,B 0,C 180,E1 26151.147,E2 26151.147} C_VEL
LIN {X 0,Y 561.356,Z 191.225,A -85,B 0,C 180,E1 26147.815,E2 26147.815} C_VEL
LIN {X 0,Y 561.396,Z 191.22,A -85,B 0,C 180,E1 26144.711,E2 26144.711} C_VEL
LIN {X 0,Y 561.348,Z 191.24,A -85,B 0,C 180,E1 26141.5,E2 26141.5} C_VEL
LIN {X 0,Y 561.392,Z 191.236,A -85,B 0,C 180,E1 26138.303,E2 26138.303} C_VEL
LIN {X 0,Y 561.36,Z 191.214,A -85,B 0,C 180,E1 26135.169,E2 26135.169} C_VEL
LIN {X 0,Y 561.351,Z 191.241,A -85,B 0,C 180,E1 26131.82,E2 26131.82} C_VEL
LIN {X 0,Y 561.41,Z 191.186,A -85,B 0,C 180,E1 26128.743,E2 26128.743} C_VEL
LIN {X 0,Y 561.35,Z 191.234,A -85,B 0,C 180,E1 26125.535,E2 26125.535} C_VEL
LIN {X 0,Y 561.362,Z 191.227,A -85,B 0,C 180,E1 26122.186,E2 26122.186} C_VEL
LIN {X 0,Y 561.382,Z 191.239,A -85,B 0,C 180,E1 26119.131,E2 26119.131} C_VEL
LIN {X 0,Y 561.348,Z 191.237,A -85,B 0,C 180,E1 26115.902,E2 26115.902} C_VEL
LIN {X 0,Y 561.408,Z 191.221,A -85,B 0,C 180,E1 26112.759,E2 26112.759} C_VEL
LIN {X 0,Y 561.357,Z 191.238,A -85,B 0,C 180,E1 26109.535,E2 26109.535} C_VEL
LIN {X 0,Y 561.353,Z 191.24,A -85,B 0,C 180,E1 26106.238,E2 26106.238} C_VEL
LIN {X 0,Y 561.404,Z 191.223,A -85,B 0,C 180,E1 26103.063,E2 26103.063} C_VEL
LIN {X 0,Y 561.346,Z 191.24,A -85,B 0,C 180,E1 26099.898,E2 26099.898} C_VEL
LIN {X 0,Y 561.374,Z 191.236,A -85,B 0,C 180,E1 26096.63,E2 26096.63} C_VEL
LIN {X 0,Y 561.365,Z 191.234,A -85,B 0,C 180,E1 26093.557,E2 26093.557} C_VEL
LIN {X 0,Y 561.348,Z 191.241,A -85,B 0,C 180,E1 26090.258,E2 26090.258} C_VEL
LIN {X 0,Y 561.409,Z 191.226,A -85,B 0,C 180,E1 26087.032,E2 26087.032} C_VEL
LIN {X 0,Y 561.347,Z 191.237,A -85,B 0,C 180,E1 26083.973,E2 26083.973} C_VEL
LIN {X 0,Y 561.363,Z 191.24,A -85,B 0,C 180,E1 26080.652,E2 26080.652} C_VEL
LIN {X 0,Y 561.384,Z 191.23,A -85,B 0,C 180,E1 26077.559,E2 26077.559} C_VEL
LIN {X 0,Y 561.346,Z 191.228,A -85,B 0,C 180,E1 26074.314,E2 26074.314} C_VEL
LIN {X 0,Y 561.398,Z 191.193,A -85,B 0,C 180,E1 26071.14,E2 26071.14} C_VEL
LIN {X 0,Y 561.353,Z 191.242,A -85,B 0,C 180,E1 26068.061,E2 26068.061} C_VEL
LIN {X 0,Y 561.343,Z 191.2,A -85,B 0,C 180,E1 26064.626,E2 26064.626} C_VEL
LIN {X 0,Y 561.423,Z 191.238,A -85,B 0,C 180,E1 26061.421,E2 26061.421} C_VEL
LIN {X 0,Y 561.35,Z 191.242,A -85,B 0,C 180,E1 26058.227,E2 26058.227} C_VEL
LIN {X 0,Y 561.356,Z 191.244,A -85,B 0,C 180,E1 26054.851,E2 26054.851} C_VEL
LIN {X 0,Y 561.419,Z 191.238,A -85,B 0,C 180,E1 26051.58,E2 26051.58} C_VEL
LIN {X 0,Y 561.348,Z 191.244,A -85,B 0,C 180,E1 26048.395,E2 26048.395} C_VEL
LIN {X 0,Y 561.368,Z 191.241,A -85,B 0,C 180,E1 26045.116,E2 26045.116} C_VEL
LIN {X 0,Y 561.378,Z 191.24,A -85,B 0,C 180,E1 26042.024,E2 26042.024} C_VEL
LIN {X 0,Y 561.348,Z 191.245,A -85,B 0,C 180,E1 26038.793,E2 26038.793} C_VEL
LIN {X 0,Y 561.41,Z 191.238,A -85,B 0,C 180,E1 26035.641,E2 26035.641} C_VEL
LIN {X 0,Y 561.353,Z 191.243,A -85,B 0,C 180,E1 26032.514,E2 26032.514} C_VEL
LIN {X 0,Y 561.356,Z 191.246,A -85,B 0,C 180,E1 26029.129,E2 26029.129} C_VEL
LIN {X 0,Y 561.41,Z 191.237,A -85,B 0,C 180,E1 26025.917,E2 26025.917} C_VEL
LIN {X 0,Y 561.345,Z 191.243,A -85,B 0,C 180,E1 26022.759,E2 26022.759} C_VEL
LIN {X 0,Y 561.35,Z 191.245,A -85,B 0,C 180,E1 26021.116,E2 26021.116} C_VEL
LIN {X 0,Y 560.364,Z 191.372,A -85,B 0,C 180,E1 26020.33,E2 26020.33} C_VEL
LIN {X 0,Y 553.913,Z 192.173,A -85,B 0,C 180,E1 26018.065,E2 26018.065} C_VEL
LIN {X 0,Y 553.438,Z 192.229,A -85,B 0,C 180,E1 26017.548,E2 26017.548} C_VEL
LIN {X 0,Y 553.426,Z 192.231,A -85,B 0,C 180,E1 26014.455,E2 26014.455} C_VEL
LIN {X 0,Y 553.409,Z 192.234,A -85,B 0,C 180,E1 26011.139,E2 26011.139} C_VEL
LIN {X 0,Y 553.471,Z 192.225,A -85,B 0,C 180,E1 26008.033,E2 26008.033} C_VEL
LIN {X 0,Y 553.412,Z 192.234,A -85,B 0,C 180,E1 26004.818,E2 26004.818} C_VEL
LIN {X 0,Y 553.412,Z 192.232,A -85,B 0,C 180,E1 26001.376,E2 26001.376} C_VEL
LIN {X 0,Y 553.471,Z 192.226,A -85,B 0,C 180,E1 25998.117,E2 25998.117} C_VEL
LIN {X 0,Y 553.412,Z 192.235,A -85,B 0,C 180,E1 25994.922,E2 25994.922} C_VEL
LIN {X 0,Y 553.413,Z 192.232,A -85,B 0,C 180,E1 25991.461,E2 25991.461} C_VEL
LIN {X 0,Y 553.48,Z 192.228,A -85,B 0,C 180,E1 25988.213,E2 25988.213} C_VEL
LIN {X 0,Y 553.415,Z 192.232,A -85,B 0,C 180,E1 25984.993,E2 25984.993} C_VEL
LIN {X 0,Y 553.415,Z 192.234,A -85,B 0,C 180,E1 25981.63,E2 25981.63} C_VEL
LIN {X 0,Y 553.465,Z 192.229,A -85,B 0,C 180,E1 25978.509,E2 25978.509} C_VEL
LIN {X 0,Y 553.409,Z 192.233,A -85,B 0,C 180,E1 25975.295,E2 25975.295} C_VEL
LIN {X 0,Y 553.432,Z 192.231,A -85,B 0,C 180,E1 25971.974,E2 25971.974} C_VEL
LIN {X 0,Y 553.435,Z 192.229,A -85,B 0,C 180,E1 25968.885,E2 25968.885} C_VEL
LIN {X 0,Y 553.409,Z 192.233,A -85,B 0,C 180,E1 25965.643,E2 25965.643} C_VEL
LIN {X 0,Y 553.464,Z 192.229,A -85,B 0,C 180,E1 25962.371,E2 25962.371} C_VEL
LIN {X 0,Y 553.418,Z 192.231,A -85,B 0,C 180,E1 25959.225,E2 25959.225} C_VEL
LIN {X 0,Y 553.405,Z 192.191,A -85,B 0,C 180,E1 25955.832,E2 25955.832} C_VEL
LIN {X 0,Y 553.472,Z 192.219,A -85,B 0,C 180,E1 25952.572,E2 25952.572} C_VEL
LIN {X 0,Y 553.409,Z 192.202,A -85,B 0,C 180,E1 25949.436,E2 25949.436} C_VEL
LIN {X 0,Y 553.414,Z 192.202,A -85,B 0,C 180,E1 25946.043,E2 25946.043} C_VEL
LIN {X 0,Y 553.473,Z 192.222,A -85,B 0,C 180,E1 25942.856,E2 25942.856} C_VEL
LIN {X 0,Y 553.409,Z 192.229,A -85,B 0,C 180,E1 25939.637,E2 25939.637} C_VEL
LIN {X 0,Y 553.431,Z 192.219,A -85,B 0,C 180,E1 25936.371,E2 25936.371} C_VEL
LIN {X 0,Y 553.425,Z 192.226,A -85,B 0,C 180,E1 25933.371,E2 25933.371} C_VEL
LIN {X 0,Y 553.411,Z 192.229,A -85,B 0,C 180,E1 25930.082,E2 25930.082} C_VEL
LIN {X 0,Y 553.474,Z 192.211,A -85,B 0,C 180,E1 25926.848,E2 25926.848} C_VEL
LIN {X 0,Y 553.416,Z 192.228,A -85,B 0,C 180,E1 25923.626,E2 25923.626} C_VEL
LIN {X 0,Y 553.41,Z 192.229,A -85,B 0,C 180,E1 25920.207,E2 25920.207} C_VEL
LIN {X 0,Y 553.468,Z 192.209,A -85,B 0,C 180,E1 25916.997,E2 25916.997} C_VEL
LIN {X 0,Y 553.416,Z 192.227,A -85,B 0,C 180,E1 25913.777,E2 25913.777} C_VEL
LIN {X 0,Y 553.411,Z 192.227,A -85,B 0,C 180,E1 25910.327,E2 25910.327} C_VEL
LIN {X 0,Y 553.47,Z 192.211,A -85,B 0,C 180,E1 25907.055,E2 25907.055} C_VEL
LIN {X 0,Y 553.412,Z 192.229,A -85,B 0,C 180,E1 25903.952,E2 25903.952} C_VEL
LIN {X 0,Y 553.418,Z 192.23,A -85,B 0,C 180,E1 25900.561,E2 25900.561} C_VEL
LIN {X 0,Y 553.471,Z 192.213,A -85,B 0,C 180,E1 25897.368,E2 25897.368} C_VEL
LIN {X 0,Y 553.411,Z 192.222,A -85,B 0,C 180,E1 25894.112,E2 25894.112} C_VEL
LIN {X 0,Y 553.418,Z 192.187,A -85,B 0,C 180,E1 25890.755,E2 25890.755} C_VEL
LIN {X 0,Y 553.45,Z 192.23,A -85,B 0,C 180,E1 25887.672,E2 25887.672} C_VEL
LIN {X 0,Y 553.407,Z 192.208,A -85,B 0,C 180,E1 25884.384,E2 25884.384} C_VEL
LIN {X 0,Y 553.446,Z 192.214,A -85,B 0,C 180,E1 25881.129,E2 25881.129} C_VEL
LIN {X 0,Y 553.424,Z 192.23,A -85,B 0,C 180,E1 25878.049,E2 25878.049} C_VEL
LIN {X 0,Y 553.413,Z 192.221,A -85,B 0,C 180,E1 25874.76,E2 25874.76} C_VEL
LIN {X 0,Y 553.477,Z 192.21,A -85,B 0,C 180,E1 25871.523,E2 25871.523} C_VEL
LIN {X 0,Y 553.49,Z 192.464,A -85,B 0,C 180,E1 25869.33,E2 25869.33} C_VEL
LIN {X 0,Y 559.841,Z 211.838,A -85,B 0,C 180,E1 25866.616,E2 25866.616} C_VEL
LIN {X 0,Y 562.96,Z 222.004,A -85,B 0,C 180,E1 25865.3,E2 25865.3} C_VEL
LIN {X 0,Y 572.633,Z 241.547,A -85,B 0,C 180,E1 25864.318,E2 25864.318} C_VEL
LIN {X 0,Y 577.5,Z 265.368,A -85,B 0,C 180,E1 25863.642,E2 25863.642} C_VEL
LIN {X 0,Y 572.512,Z 522.163,A -85,B 0,C 180,E1 25860.23,E2 25860.23} C_VEL
LIN {X 0,Y 571.787,Z 539.756,A -85,B 0,C 180,E1 25859.906,E2 25859.906} C_VEL
LIN {X 0,Y 570.835,Z 556.853,A -85,B 0,C 180,E1 25859.481,E2 25859.481} C_VEL
LIN {X 0,Y 569.695,Z 573.909,A -85,B 0,C 180,E1 25858.941,E2 25858.941} C_VEL
LIN {X 0,Y 568.287,Z 591.796,A -85,B 0,C 180,E1 25858.244,E2 25858.244} C_VEL
LIN {X 0,Y 566.377,Z 613.428,A -85,B 0,C 180,E1 25857.205,E2 25857.205} C_VEL
LIN {X 0,Y 564.573,Z 631.18,A -85,B 0,C 180,E1 25856.163,E2 25856.163} C_VEL
LIN {X 0,Y 562.932,Z 646.552,A -85,B 0,C 180,E1 25855.116,E2 25855.116} C_VEL
LIN {X 0,Y 561.366,Z 660.726,A -85,B 0,C 180,E1 25854.013,E2 25854.013} C_VEL
LIN {X 0,Y 559.831,Z 674.437,A -85,B 0,C 180,E1 25852.8,E2 25852.8} C_VEL
LIN {X 0,Y 558.412,Z 687.113,A -85,B 0,C 180,E1 25851.532,E2 25851.532} C_VEL
LIN {X 0,Y 557.06,Z 699.298,A -85,B 0,C 180,E1 25850.156,E2 25850.156} C_VEL
LIN {X 0,Y 555.737,Z 711.998,A -85,B 0,C 180,E1 25848.524,E2 25848.524} C_VEL
LIN {X 0,Y 554.339,Z 726.427,A -85,B 0,C 180,E1 25846.341,E2 25846.341} C_VEL
LIN {X 0,Y 553.48,Z 736.459,A -85,B 0,C 180,E1 25844.541,E2 25844.541} C_VEL
LIN {X 0,Y 552.896,Z 744.581,A -85,B 0,C 180,E1 25842.851,E2 25842.851} C_VEL
LIN {X 0,Y 552.48,Z 751.518,A -85,B 0,C 180,E1 25841.164,E2 25841.164} C_VEL
LIN {X 0,Y 552.206,Z 757.356,A -85,B 0,C 180,E1 25839.483,E2 25839.483} C_VEL
LIN {X 0,Y 552.033,Z 762.429,A -85,B 0,C 180,E1 25837.702,E2 25837.702} C_VEL
LIN {X 0,Y 551.957,Z 766.396,A -85,B 0,C 180,E1 25835.926,E2 25835.926} C_VEL
LIN {X 0,Y 551.927,Z 769.447,A -85,B 0,C 180,E1 25834.051,E2 25834.051} C_VEL
LIN {X 0,Y 551.921,Z 771.691,A -85,B 0,C 180,E1 25831.765,E2 25831.765} C_VEL
LIN {X 0,Y 551.916,Z 772.058,A -85,B 0,C 180,E1 25829.481,E2 25829.481} C_VEL
LIN {X 0,Y 551.919,Z 771.171,A -85,B 0,C 180,E1 25827.612,E2 25827.612} C_VEL
LIN {X 0,Y 551.929,Z 769.153,A -85,B 0,C 180,E1 25825.741,E2 25825.741} C_VEL
LIN {X 0,Y 551.963,Z 766.188,A -85,B 0,C 180,E1 25823.97,E2 25823.97} C_VEL
LIN {X 0,Y 552.04,Z 762.159,A -85,B 0,C 180,E1 25822.194,E2 25822.194} C_VEL
LIN {X 0,Y 552.216,Z 757.022,A -85,B 0,C 180,E1 25820.412,E2 25820.412} C_VEL
LIN {X 0,Y 552.519,Z 750.72,A -85,B 0,C 180,E1 25818.625,E2 25818.625} C_VEL
LIN {X 0,Y 553.026,Z 742.707,A -85,B 0,C 180,E1 25816.727,E2 25816.727} C_VEL
LIN {X 0,Y 553.961,Z 730.758,A -85,B 0,C 180,E1 25814.401,E2 25814.401} C_VEL
LIN {X 0,Y 554.892,Z 720.415,A -85,B 0,C 180,E1 25812.706,E2 25812.706} C_VEL
LIN {X 0,Y 555.997,Z 709.306,A -85,B 0,C 180,E1 25811.115,E2 25811.115} C_VEL
LIN {X 0,Y 557.159,Z 698.402,A -85,B 0,C 180,E1 25809.738,E2 25809.738} C_VEL
LIN {X 0,Y 558.524,Z 686.113,A -85,B 0,C 180,E1 25808.362,E2 25808.362} C_VEL
LIN {X 0,Y 560.017,Z 672.754,A -85,B 0,C 180,E1 25807.041,E2 25807.041} C_VEL
LIN {X 0,Y 561.892,Z 656.311,A -85,B 0,C 180,E1 25805.62,E2 25805.62} C_VEL
LIN {X 0,Y 563.985,Z 636.825,A -85,B 0,C 180,E1 25804.203,E2 25804.203} C_VEL
LIN {X 0,Y 565.608,Z 620.794,A -85,B 0,C 180,E1 25803.209,E2 25803.209} C_VEL
LIN {X 0,Y 567.107,Z 605.204,A -85,B 0,C 180,E1 25802.378,E2 25802.378} C_VEL
LIN {X 0,Y 568.489,Z 589.307,A -85,B 0,C 180,E1 25801.652,E2 25801.652} C_VEL
LIN {X 0,Y 569.75,Z 573.165,A -85,B 0,C 180,E1 25801.033,E2 25801.033} C_VEL
LIN {X 0,Y 570.887,Z 556.051,A -85,B 0,C 180,E1 25800.496,E2 25800.496} C_VEL
LIN {X 0,Y 571.838,Z 538.797,A -85,B 0,C 180,E1 25800.073,E2 25800.073} C_VEL
LIN {X 0,Y 572.573,Z 520.313,A -85,B 0,C 180,E1 25799.741,E2 25799.741} C_VEL
LIN {X 0,Y 577.504,Z 264.46,A -85,B 0,C 180,E1 25796.345,E2 25796.345} C_VEL
LIN {X 0,Y 572.129,Z 240.168,A -85,B 0,C 180,E1 25795.627,E2 25795.627} C_VEL
LIN {X 0,Y 562.959,Z 222.003,A -85,B 0,C 180,E1 25794.7,E2 25794.7} C_VEL
LIN {X 0,Y 557.583,Z 204.867,A -85,B 0,C 180,E1 25792.432,E2 25792.432} C_VEL
LIN {X 0,Y 553.473,Z 192.334,A -85,B 0,C 180,E1 25790.633,E2 25790.633} C_VEL
LIN {X 0,Y 553.407,Z 192.216,A -85,B 0,C 180,E1 25787.491,E2 25787.491} C_VEL
LIN {X 0,Y 553.462,Z 192.205,A -85,B 0,C 180,E1 25784.331,E2 25784.331} C_VEL
LIN {X 0,Y 553.416,Z 192.222,A -85,B 0,C 180,E1 25781.26,E2 25781.26} C_VEL
LIN {X 0,Y 553.417,Z 192.232,A -85,B 0,C 180,E1 25777.866,E2 25777.866} C_VEL
LIN {X 0,Y 553.467,Z 192.196,A -85,B 0,C 180,E1 25774.686,E2 25774.686} C_VEL
LIN {X 0,Y 553.412,Z 192.23,A -85,B 0,C 180,E1 25771.477,E2 25771.477} C_VEL
LIN {X 0,Y 553.42,Z 192.177,A -85,B 0,C 180,E1 25768.136,E2 25768.136} C_VEL
LIN {X 0,Y 553.459,Z 192.222,A -85,B 0,C 180,E1 25764.933,E2 25764.933} C_VEL
LIN {X 0,Y 553.405,Z 192.217,A -85,B 0,C 180,E1 25761.74,E2 25761.74} C_VEL
LIN {X 0,Y 553.449,Z 192.214,A -85,B 0,C 180,E1 25758.493,E2 25758.493} C_VEL
LIN {X 0,Y 553.431,Z 192.226,A -85,B 0,C 180,E1 25755.295,E2 25755.295} C_VEL
LIN {X 0,Y 553.409,Z 192.222,A -85,B 0,C 180,E1 25751.992,E2 25751.992} C_VEL
LIN {X 0,Y 553.461,Z 192.21,A -85,B 0,C 180,E1 25748.729,E2 25748.729} C_VEL
LIN {X 0,Y 553.416,Z 192.229,A -85,B 0,C 180,E1 25745.599,E2 25745.599} C_VEL
LIN {X 0,Y 553.411,Z 192.222,A -85,B 0,C 180,E1 25742.175,E2 25742.175} C_VEL
LIN {X 0,Y 553.476,Z 192.215,A -85,B 0,C 180,E1 25738.965,E2 25738.965} C_VEL
LIN {X 0,Y 553.415,Z 192.228,A -85,B 0,C 180,E1 25735.709,E2 25735.709} C_VEL
LIN {X 0,Y 553.411,Z 192.219,A -85,B 0,C 180,E1 25732.316,E2 25732.316} C_VEL
LIN {X 0,Y 553.469,Z 192.22,A -85,B 0,C 180,E1 25729.171,E2 25729.171} C_VEL
LIN {X 0,Y 553.409,Z 192.228,A -85,B 0,C 180,E1 25725.956,E2 25725.956} C_VEL
LIN {X 0,Y 553.425,Z 192.219,A -85,B 0,C 180,E1 25722.656,E2 25722.656} C_VEL
LIN {X 0,Y 553.452,Z 192.222,A -85,B 0,C 180,E1 25719.483,E2 25719.483} C_VEL
LIN {X 0,Y 553.408,Z 192.23,A -85,B 0,C 180,E1 25716.336,E2 25716.336} C_VEL
LIN {X 0,Y 553.461,Z 192.176,A -85,B 0,C 180,E1 25713.15,E2 25713.15} C_VEL
LIN {X 0,Y 553.416,Z 192.217,A -85,B 0,C 180,E1 25709.969,E2 25709.969} C_VEL
LIN {X 0,Y 553.409,Z 192.216,A -85,B 0,C 180,E1 25706.576,E2 25706.576} C_VEL
LIN {X 0,Y 553.465,Z 192.2,A -85,B 0,C 180,E1 25703.324,E2 25703.324} C_VEL
LIN {X 0,Y 553.41,Z 192.231,A -85,B 0,C 180,E1 25700.238,E2 25700.238} C_VEL
LIN {X 0,Y 553.422,Z 192.232,A -85,B 0,C 180,E1 25696.872,E2 25696.872} C_VEL
LIN {X 0,Y 553.465,Z 192.227,A -85,B 0,C 180,E1 25693.632,E2 25693.632} C_VEL
LIN {X 0,Y 553.409,Z 192.231,A -85,B 0,C 180,E1 25690.432,E2 25690.432} C_VEL
LIN {X 0,Y 553.436,Z 192.231,A -85,B 0,C 180,E1 25687.179,E2 25687.179} C_VEL
LIN {X 0,Y 553.442,Z 192.231,A -85,B 0,C 180,E1 25683.976,E2 25683.976} C_VEL
LIN {X 0,Y 553.407,Z 192.231,A -85,B 0,C 180,E1 25680.747,E2 25680.747} C_VEL
LIN {X 0,Y 553.466,Z 192.228,A -85,B 0,C 180,E1 25677.544,E2 25677.544} C_VEL
LIN {X 0,Y 553.422,Z 192.234,A -85,B 0,C 180,E1 25674.323,E2 25674.323} C_VEL
LIN {X 0,Y 553.411,Z 192.232,A -85,B 0,C 180,E1 25670.959,E2 25670.959} C_VEL
LIN {X 0,Y 553.473,Z 192.228,A -85,B 0,C 180,E1 25667.774,E2 25667.774} C_VEL
LIN {X 0,Y 553.41,Z 192.234,A -85,B 0,C 180,E1 25664.65,E2 25664.65} C_VEL
LIN {X 0,Y 553.425,Z 192.231,A -85,B 0,C 180,E1 25661.356,E2 25661.356} C_VEL
LIN {X 0,Y 553.447,Z 192.231,A -85,B 0,C 180,E1 25658.205,E2 25658.205} C_VEL
LIN {X 0,Y 553.438,Z 192.229,A -85,B 0,C 180,E1 25657.548,E2 25657.548} C_VEL
LIN {X 0,Y 552.645,Z 192.894,A -85,B 0,C 180,E1 25656.751,E2 25656.751} C_VEL
LIN {X 0,Y 548.028,Z 197.345,A -85,B 0,C 180,E1 25654.519,E2 25654.519} C_VEL
LIN {X 0,Y 547.754,Z 197.829,A -85,B 0,C 180,E1 25653.94,E2 25653.94} C_VEL
LIN {X 0,Y 548.396,Z 198.456,A -85,B 0,C 180,E1 25651.463,E2 25651.463} C_VEL
LIN {X 0,Y 548.424,Z 198.493,A -85,B 0,C 180,E1 25648.955,E2 25648.955} C_VEL
LIN {X 0,Y 547.883,Z 198,A -85,B 0,C 180,E1 25646.548,E2 25646.548} C_VEL
LIN {X 0,Y 546.891,Z 196.792,A -85,B 0,C 180,E1 25644.23,E2 25644.23} C_VEL
LIN {X 0,Y 546.029,Z 195.301,A -85,B 0,C 180,E1 25642.742,E2 25642.742} C_VEL
LIN {X 0,Y 545.521,Z 193.577,A -85,B 0,C 180,E1 25641.145,E2 25641.145} C_VEL
LIN {X 0,Y 545.492,Z 193.218,A -85,B 0,C 180,E1 25638.584,E2 25638.584} C_VEL
LIN {X 0,Y 545.472,Z 193.223,A -85,B 0,C 180,E1 25635.349,E2 25635.349} C_VEL
LIN {X 0,Y 545.535,Z 193.216,A -85,B 0,C 180,E1 25632.179,E2 25632.179} C_VEL
LIN {X 0,Y 545.478,Z 193.22,A -85,B 0,C 180,E1 25628.912,E2 25628.912} C_VEL
LIN {X 0,Y 545.475,Z 193.224,A -85,B 0,C 180,E1 25625.53,E2 25625.53} C_VEL
LIN {X 0,Y 545.539,Z 193.214,A -85,B 0,C 180,E1 25622.259,E2 25622.259} C_VEL
LIN {X 0,Y 545.474,Z 193.22,A -85,B 0,C 180,E1 25619.079,E2 25619.079} C_VEL
LIN {X 0,Y 545.475,Z 193.222,A -85,B 0,C 180,E1 25615.632,E2 25615.632} C_VEL
LIN {X 0,Y 545.532,Z 193.215,A -85,B 0,C 180,E1 25612.354,E2 25612.354} C_VEL
LIN {X 0,Y 545.479,Z 193.219,A -85,B 0,C 180,E1 25609.133,E2 25609.133} C_VEL
LIN {X 0,Y 545.473,Z 193.222,A -85,B 0,C 180,E1 25605.709,E2 25605.709} C_VEL
LIN {X 0,Y 545.528,Z 193.217,A -85,B 0,C 180,E1 25602.416,E2 25602.416} C_VEL
LIN {X 0,Y 545.479,Z 193.22,A -85,B 0,C 180,E1 25599.228,E2 25599.228} C_VEL
LIN {X 0,Y 545.469,Z 193.179,A -85,B 0,C 180,E1 25595.893,E2 25595.893} C_VEL
LIN {X 0,Y 545.533,Z 193.207,A -85,B 0,C 180,E1 25592.606,E2 25592.606} C_VEL
LIN {X 0,Y 545.471,Z 193.188,A -85,B 0,C 180,E1 25589.424,E2 25589.424} C_VEL
LIN {X 0,Y 545.472,Z 193.191,A -85,B 0,C 180,E1 25585.983,E2 25585.983} C_VEL
LIN {X 0,Y 545.544,Z 193.207,A -85,B 0,C 180,E1 25582.751,E2 25582.751} C_VEL
LIN {X 0,Y 545.477,Z 193.218,A -85,B 0,C 180,E1 25579.488,E2 25579.488} C_VEL
LIN {X 0,Y 545.472,Z 193.213,A -85,B 0,C 180,E1 25576.069,E2 25576.069} C_VEL
LIN {X 0,Y 545.534,Z 193.199,A -85,B 0,C 180,E1 25572.852,E2 25572.852} C_VEL
LIN {X 0,Y 545.478,Z 193.218,A -85,B 0,C 180,E1 25569.583,E2 25569.583} C_VEL
LIN {X 0,Y 545.472,Z 193.215,A -85,B 0,C 180,E1 25566.209,E2 25566.209} C_VEL
LIN {X 0,Y 545.528,Z 193.2,A -85,B 0,C 180,E1 25562.942,E2 25562.942} C_VEL
LIN {X 0,Y 545.471,Z 193.218,A -85,B 0,C 180,E1 25559.79,E2 25559.79} C_VEL
LIN {X 0,Y 545.474,Z 193.209,A -85,B 0,C 180,E1 25556.321,E2 25556.321} C_VEL
LIN {X 0,Y 545.542,Z 193.198,A -85,B 0,C 180,E1 25553.052,E2 25553.052} C_VEL
LIN {X 0,Y 545.48,Z 193.216,A -85,B 0,C 180,E1 25549.758,E2 25549.758} C_VEL
LIN {X 0,Y 545.475,Z 193.211,A -85,B 0,C 180,E1 25546.43,E2 25546.43} C_VEL
LIN {X 0,Y 545.531,Z 193.204,A -85,B 0,C 180,E1 25543.276,E2 25543.276} C_VEL
LIN {X 0,Y 545.472,Z 193.219,A -85,B 0,C 180,E1 25540.065,E2 25540.065} C_VEL
LIN {X 0,Y 545.485,Z 193.218,A -85,B 0,C 180,E1 25536.667,E2 25536.667} C_VEL
LIN {X 0,Y 545.526,Z 193.181,A -85,B 0,C 180,E1 25533.422,E2 25533.422} C_VEL
LIN {X 0,Y 545.468,Z 193.189,A -85,B 0,C 180,E1 25530.213,E2 25530.213} C_VEL
LIN {X 0,Y 545.49,Z 193.21,A -85,B 0,C 180,E1 25526.885,E2 25526.885} C_VEL
LIN {X 0,Y 545.51,Z 193.201,A -85,B 0,C 180,E1 25523.698,E2 25523.698} C_VEL
LIN {X 0,Y 545.467,Z 193.198,A -85,B 0,C 180,E1 25520.499,E2 25520.499} C_VEL
LIN {X 0,Y 545.522,Z 193.212,A -85,B 0,C 180,E1 25517.298,E2 25517.298} C_VEL
LIN {X 0,Y 545.493,Z 193.22,A -85,B 0,C 180,E1 25513.996,E2 25513.996} C_VEL
LIN {X 0,Y 545.475,Z 193.222,A -85,B 0,C 180,E1 25510.729,E2 25510.729} C_VEL
LIN {X 0,Y 545.562,Z 193.543,A -85,B 0,C 180,E1 25509.849,E2 25509.849} C_VEL
LIN {X 0,Y 551.675,Z 212.02,A -85,B 0,C 180,E1 25507.195,E2 25507.195} C_VEL
LIN {X 0,Y 554.535,Z 221.272,A -85,B 0,C 180,E1 25505.943,E2 25505.943} C_VEL
LIN {X 0,Y 564.711,Z 241.325,A -85,B 0,C 180,E1 25504.868,E2 25504.868} C_VEL
LIN {X 0,Y 566.522,Z 245.577,A -85,B 0,C 180,E1 25504.677,E2 25504.677} C_VEL
LIN {X 0,Y 570.803,Z 266.86,A -85,B 0,C 180,E1 25504.066,E2 25504.066} C_VEL
LIN {X 0,Y 565.588,Z 522.296,A -85,B 0,C 180,E1 25500.634,E2 25500.634} C_VEL
LIN {X 0,Y 564.83,Z 539.888,A -85,B 0,C 180,E1 25500.305,E2 25500.305} C_VEL
LIN {X 0,Y 563.825,Z 557.089,A -85,B 0,C 180,E1 25499.872,E2 25499.872} C_VEL
LIN {X 0,Y 562.651,Z 573.859,A -85,B 0,C 180,E1 25499.334,E2 25499.334} C_VEL
LIN {X 0,Y 561.187,Z 591.62,A -85,B 0,C 180,E1 25498.635,E2 25498.635} C_VEL
LIN {X 0,Y 559.185,Z 613.251,A -85,B 0,C 180,E1 25497.585,E2 25497.585} C_VEL
LIN {X 0,Y 557.298,Z 631.003,A -85,B 0,C 180,E1 25496.531,E2 25496.531} C_VEL
LIN {X 0,Y 555.578,Z 646.374,A -85,B 0,C 180,E1 25495.472,E2 25495.472} C_VEL
LIN {X 0,Y 553.928,Z 660.548,A -85,B 0,C 180,E1 25494.356,E2 25494.356} C_VEL
LIN {X 0,Y 552.296,Z 674.376,A -85,B 0,C 180,E1 25493.118,E2 25493.118} C_VEL
LIN {X 0,Y 550.759,Z 687.434,A -85,B 0,C 180,E1 25491.79,E2 25491.79} C_VEL
LIN {X 0,Y 549.291,Z 700.004,A -85,B 0,C 180,E1 25490.343,E2 25490.343} C_VEL
LIN {X 0,Y 547.704,Z 714.623,A -85,B 0,C 180,E1 25488.408,E2 25488.408} C_VEL
LIN {X 0,Y 546.441,Z 726.868,A -85,B 0,C 180,E1 25486.474,E2 25486.474} C_VEL
LIN {X 0,Y 545.589,Z 736.281,A -85,B 0,C 180,E1 25484.756,E2 25484.756} C_VEL
LIN {X 0,Y 544.96,Z 744.484,A -85,B 0,C 180,E1 25483.022,E2 25483.022} C_VEL
LIN {X 0,Y 544.513,Z 751.426,A -85,B 0,C 180,E1 25481.307,E2 25481.307} C_VEL
LIN {X 0,Y 544.212,Z 757.512,A -85,B 0,C 180,E1 25479.517,E2 25479.517} C_VEL
LIN {X 0,Y 544.03,Z 762.792,A -85,B 0,C 180,E1 25477.603,E2 25477.603} C_VEL
LIN {X 0,Y 543.932,Z 767.647,A -85,B 0,C 180,E1 25475.273,E2 25475.273} C_VEL
LIN {X 0,Y 543.914,Z 770.467,A -85,B 0,C 180,E1 25473.056,E2 25473.056} C_VEL
LIN {X 0,Y 543.919,Z 771.708,A -85,B 0,C 180,E1 25471.159,E2 25471.159} C_VEL
LIN {X 0,Y 543.92,Z 771.854,A -85,B 0,C 180,E1 25469.368,E2 25469.368} C_VEL
LIN {X 0,Y 543.921,Z 770.996,A -85,B 0,C 180,E1 25467.577,E2 25467.577} C_VEL
LIN {X 0,Y 543.929,Z 768.977,A -85,B 0,C 180,E1 25465.678,E2 25465.678} C_VEL
LIN {X 0,Y 543.968,Z 766.013,A -85,B 0,C 180,E1 25463.881,E2 25463.881} C_VEL
LIN {X 0,Y 544.05,Z 761.983,A -85,B 0,C 180,E1 25462.078,E2 25462.078} C_VEL
LIN {X 0,Y 544.236,Z 756.846,A -85,B 0,C 180,E1 25460.27,E2 25460.27} C_VEL
LIN {X 0,Y 544.561,Z 750.542,A -85,B 0,C 180,E1 25458.457,E2 25458.457} C_VEL
LIN {X 0,Y 545.1,Z 742.529,A -85,B 0,C 180,E1 25456.531,E2 25456.531} C_VEL
LIN {X 0,Y 546.099,Z 730.579,A -85,B 0,C 180,E1 25454.17,E2 25454.17} C_VEL
LIN {X 0,Y 547.092,Z 720.237,A -85,B 0,C 180,E1 25452.451,E2 25452.451} C_VEL
LIN {X 0,Y 548.264,Z 709.127,A -85,B 0,C 180,E1 25450.839,E2 25450.839} C_VEL
LIN {X 0,Y 549.498,Z 698.223,A -85,B 0,C 180,E1 25449.443,E2 25449.443} C_VEL
LIN {X 0,Y 550.954,Z 685.769,A -85,B 0,C 180,E1 25448.031,E2 25448.031} C_VEL
LIN {X 0,Y 552.51,Z 672.576,A -85,B 0,C 180,E1 25446.711,E2 25446.711} C_VEL
LIN {X 0,Y 554.486,Z 656.133,A -85,B 0,C 180,E1 25445.273,E2 25445.273} C_VEL
LIN {X 0,Y 556.678,Z 636.647,A -85,B 0,C 180,E1 25443.839,E2 25443.839} C_VEL
LIN {X 0,Y 558.385,Z 620.617,A -85,B 0,C 180,E1 25442.835,E2 25442.835} C_VEL
LIN {X 0,Y 559.956,Z 605.028,A -85,B 0,C 180,E1 25441.994,E2 25441.994} C_VEL
LIN {X 0,Y 561.402,Z 589.13,A -85,B 0,C 180,E1 25441.261,E2 25441.261} C_VEL
LIN {X 0,Y 562.718,Z 572.989,A -85,B 0,C 180,E1 25440.636,E2 25440.636} C_VEL
LIN {X 0,Y 563.891,Z 556.104,A -85,B 0,C 180,E1 25440.101,E2 25440.101} C_VEL
LIN {X 0,Y 564.88,Z 538.963,A -85,B 0,C 180,E1 25439.675,E2 25439.675} C_VEL
LIN {X 0,Y 565.634,Z 520.96,A -85,B 0,C 180,E1 25439.345,E2 25439.345} C_VEL
LIN {X 0,Y 570.81,Z 265.938,A -85,B 0,C 180,E1 25435.921,E2 25435.921} C_VEL
LIN {X 0,Y 565.97,Z 243.902,A -85,B 0,C 180,E1 25435.259,E2 25435.259} C_VEL
LIN {X 0,Y 556.143,Z 224.67,A -85,B 0,C 180,E1 25434.259,E2 25434.259} C_VEL
LIN {X 0,Y 554.422,Z 220.941,A -85,B 0,C 180,E1 25434.024,E2 25434.024} C_VEL
LIN {X 0,Y 548.215,Z 201.494,A -85,B 0,C 180,E1 25431.319,E2 25431.319} C_VEL
LIN {X 0,Y 545.523,Z 193.335,A -85,B 0,C 180,E1 25430.102,E2 25430.102} C_VEL
LIN {X 0,Y 545.488,Z 193.208,A -85,B 0,C 180,E1 25427.002,E2 25427.002} C_VEL
LIN {X 0,Y 545.471,Z 193.205,A -85,B 0,C 180,E1 25423.617,E2 25423.617} C_VEL
LIN {X 0,Y 545.533,Z 193.189,A -85,B 0,C 180,E1 25420.454,E2 25420.454} C_VEL
LIN {X 0,Y 545.478,Z 193.221,A -85,B 0,C 180,E1 25417.304,E2 25417.304} C_VEL
LIN {X 0,Y 545.473,Z 193.202,A -85,B 0,C 180,E1 25413.866,E2 25413.866} C_VEL
LIN {X 0,Y 545.543,Z 193.197,A -85,B 0,C 180,E1 25410.633,E2 25410.633} C_VEL
LIN {X 0,Y 545.472,Z 193.173,A -85,B 0,C 180,E1 25407.394,E2 25407.394} C_VEL
LIN {X 0,Y 545.477,Z 193.218,A -85,B 0,C 180,E1 25404.013,E2 25404.013} C_VEL
LIN {X 0,Y 545.535,Z 193.206,A -85,B 0,C 180,E1 25400.829,E2 25400.829} C_VEL
LIN {X 0,Y 545.472,Z 193.202,A -85,B 0,C 180,E1 25397.605,E2 25397.605} C_VEL
LIN {X 0,Y 545.476,Z 193.21,A -85,B 0,C 180,E1 25394.174,E2 25394.174} C_VEL
LIN {X 0,Y 545.526,Z 193.211,A -85,B 0,C 180,E1 25390.989,E2 25390.989} C_VEL
LIN {X 0,Y 545.468,Z 193.2,A -85,B 0,C 180,E1 25387.796,E2 25387.796} C_VEL
LIN {X 0,Y 545.495,Z 193.212,A -85,B 0,C 180,E1 25384.521,E2 25384.521} C_VEL
LIN {X 0,Y 545.51,Z 193.211,A -85,B 0,C 180,E1 25381.26,E2 25381.26} C_VEL
LIN {X 0,Y 545.466,Z 193.202,A -85,B 0,C 180,E1 25378.004,E2 25378.004} C_VEL
LIN {X 0,Y 545.507,Z 193.214,A -85,B 0,C 180,E1 25374.742,E2 25374.742} C_VEL
LIN {X 0,Y 545.481,Z 193.209,A -85,B 0,C 180,E1 25371.674,E2 25371.674} C_VEL
LIN {X 0,Y 545.472,Z 193.205,A -85,B 0,C 180,E1 25368.367,E2 25368.367} C_VEL
LIN {X 0,Y 545.543,Z 193.215,A -85,B 0,C 180,E1 25365.132,E2 25365.132} C_VEL
LIN {X 0,Y 545.479,Z 193.212,A -85,B 0,C 180,E1 25361.843,E2 25361.843} C_VEL
LIN {X 0,Y 545.473,Z 193.205,A -85,B 0,C 180,E1 25358.493,E2 25358.493} C_VEL
LIN {X 0,Y 545.533,Z 193.207,A -85,B 0,C 180,E1 25355.298,E2 25355.298} C_VEL
LIN {X 0,Y 545.472,Z 193.161,A -85,B 0,C 180,E1 25352.013,E2 25352.013} C_VEL
LIN {X 0,Y 545.475,Z 193.221,A -85,B 0,C 180,E1 25348.628,E2 25348.628} C_VEL
LIN {X 0,Y 545.525,Z 193.169,A -85,B 0,C 180,E1 25345.372,E2 25345.372} C_VEL
LIN {X 0,Y 545.475,Z 193.218,A -85,B 0,C 180,E1 25342.115,E2 25342.115} C_VEL
LIN {X 0,Y 545.476,Z 193.22,A -85,B 0,C 180,E1 25338.707,E2 25338.707} C_VEL
LIN {X 0,Y 545.532,Z 193.217,A -85,B 0,C 180,E1 25335.471,E2 25335.471} C_VEL
LIN {X 0,Y 545.477,Z 193.22,A -85,B 0,C 180,E1 25332.221,E2 25332.221} C_VEL
LIN {X 0,Y 545.473,Z 193.222,A -85,B 0,C 180,E1 25328.816,E2 25328.816} C_VEL
LIN {X 0,Y 545.531,Z 193.218,A -85,B 0,C 180,E1 25325.646,E2 25325.646} C_VEL
LIN {X 0,Y 545.472,Z 193.222,A -85,B 0,C 180,E1 25322.481,E2 25322.481} C_VEL
LIN {X 0,Y 545.489,Z 193.219,A -85,B 0,C 180,E1 25319.177,E2 25319.177} C_VEL
LIN {X 0,Y 545.502,Z 193.219,A -85,B 0,C 180,E1 25316.083,E2 25316.083} C_VEL
LIN {X 0,Y 545.47,Z 193.223,A -85,B 0,C 180,E1 25312.865,E2 25312.865} C_VEL
LIN {X 0,Y 545.532,Z 193.214,A -85,B 0,C 180,E1 25309.706,E2 25309.706} C_VEL
LIN {X 0,Y 545.477,Z 193.222,A -85,B 0,C 180,E1 25306.504,E2 25306.504} C_VEL
LIN {X 0,Y 545.476,Z 193.221,A -85,B 0,C 180,E1 25303.136,E2 25303.136} C_VEL
LIN {X 0,Y 545.536,Z 193.243,A -85,B 0,C 180,E1 25299.92,E2 25299.92} C_VEL
LIN {X 0,Y 545.739,Z 194.275,A -85,B 0,C 180,E1 25298.003,E2 25298.003} C_VEL
LIN {X 0,Y 546.594,Z 196.371,A -85,B 0,C 180,E1 25296.301,E2 25296.301} C_VEL
LIN {X 0,Y 547.595,Z 197.691,A -85,B 0,C 180,E1 25294.293,E2 25294.293} C_VEL
LIN {X 0,Y 547.754,Z 197.829,A -85,B 0,C 180,E1 25293.94,E2 25293.94} C_VEL
LIN {X 0,Y 547.883,Z 199.031,A -85,B 0,C 180,E1 25293.137,E2 25293.137} C_VEL
LIN {X 0,Y 547.575,Z 205.534,A -85,B 0,C 180,E1 25291.084,E2 25291.084} C_VEL
LIN {X 0,Y 547.497,Z 206.44,A -85,B 0,C 180,E1 25290.337,E2 25290.337} C_VEL
LIN {X 0,Y 547.279,Z 206.236,A -85,B 0,C 180,E1 25287.906,E2 25287.906} C_VEL
LIN {X 0,Y 546.507,Z 205.539,A -85,B 0,C 180,E1 25285.488,E2 25285.488} C_VEL
LIN {X 0,Y 545.397,Z 204.016,A -85,B 0,C 180,E1 25283.263,E2 25283.263} C_VEL
LIN {X 0,Y 544.089,Z 201.607,A -85,B 0,C 180,E1 25281.38,E2 25281.38} C_VEL
LIN {X 0,Y 541.968,Z 200.418,A -85,B 0,C 180,E1 25279.155,E2 25279.155} C_VEL
LIN {X 0,Y 539.547,Z 198.601,A -85,B 0,C 180,E1 25277.107,E2 25277.107} C_VEL
LIN {X 0,Y 538.196,Z 196.438,A -85,B 0,C 180,E1 25275.971,E2 25275.971} C_VEL
LIN {X 0,Y 537.593,Z 194.626,A -85,B 0,C 180,E1 25275.019,E2 25275.019} C_VEL
LIN {X 0,Y 537.532,Z 194.211,A -85,B 0,C 180,E1 25273.332,E2 25273.332} C_VEL
LIN {X 0,Y 537.588,Z 194.203,A -85,B 0,C 180,E1 25270.103,E2 25270.103} C_VEL
LIN {X 0,Y 537.541,Z 194.212,A -85,B 0,C 180,E1 25266.894,E2 25266.894} C_VEL
LIN {X 0,Y 537.534,Z 194.209,A -85,B 0,C 180,E1 25263.474,E2 25263.474} C_VEL
LIN {X 0,Y 537.593,Z 194.204,A -85,B 0,C 180,E1 25260.229,E2 25260.229} C_VEL
LIN {X 0,Y 537.543,Z 194.212,A -85,B 0,C 180,E1 25256.98,E2 25256.98} C_VEL
LIN {X 0,Y 537.535,Z 194.209,A -85,B 0,C 180,E1 25253.608,E2 25253.608} C_VEL
LIN {X 0,Y 537.597,Z 194.204,A -85,B 0,C 180,E1 25250.355,E2 25250.355} C_VEL
LIN {X 0,Y 537.542,Z 194.21,A -85,B 0,C 180,E1 25247.101,E2 25247.101} C_VEL
LIN {X 0,Y 537.538,Z 194.21,A -85,B 0,C 180,E1 25243.786,E2 25243.786} C_VEL
LIN {X 0,Y 537.598,Z 194.205,A -85,B 0,C 180,E1 25240.475,E2 25240.475} C_VEL
LIN {X 0,Y 537.541,Z 194.195,A -85,B 0,C 180,E1 25237.196,E2 25237.196} C_VEL
LIN {X 0,Y 537.529,Z 194.18,A -85,B 0,C 180,E1 25233.76,E2 25233.76} C_VEL
LIN {X 0,Y 537.587,Z 194.194,A -85,B 0,C 180,E1 25230.515,E2 25230.515} C_VEL
LIN {X 0,Y 537.534,Z 194.147,A -85,B 0,C 180,E1 25227.352,E2 25227.352} C_VEL
LIN {X 0,Y 537.533,Z 194.209,A -85,B 0,C 180,E1 25223.923,E2 25223.923} C_VEL
LIN {X 0,Y 537.594,Z 194.192,A -85,B 0,C 180,E1 25220.695,E2 25220.695} C_VEL
LIN {X 0,Y 537.542,Z 194.196,A -85,B 0,C 180,E1 25217.426,E2 25217.426} C_VEL
LIN {X 0,Y 537.533,Z 194.205,A -85,B 0,C 180,E1 25214.104,E2 25214.104} C_VEL
LIN {X 0,Y 537.59,Z 194.196,A -85,B 0,C 180,E1 25210.828,E2 25210.828} C_VEL
LIN {X 0,Y 537.539,Z 194.193,A -85,B 0,C 180,E1 25207.559,E2 25207.559} C_VEL
LIN {X 0,Y 537.532,Z 194.206,A -85,B 0,C 180,E1 25204.16,E2 25204.16} C_VEL
LIN {X 0,Y 537.587,Z 194.196,A -85,B 0,C 180,E1 25200.853,E2 25200.853} C_VEL
LIN {X 0,Y 537.54,Z 194.195,A -85,B 0,C 180,E1 25197.655,E2 25197.655} C_VEL
LIN {X 0,Y 537.532,Z 194.205,A -85,B 0,C 180,E1 25194.235,E2 25194.235} C_VEL
LIN {X 0,Y 537.59,Z 194.19,A -85,B 0,C 180,E1 25191.011,E2 25191.011} C_VEL
LIN {X 0,Y 537.542,Z 194.196,A -85,B 0,C 180,E1 25187.757,E2 25187.757} C_VEL
LIN {X 0,Y 537.534,Z 194.207,A -85,B 0,C 180,E1 25184.352,E2 25184.352} C_VEL
LIN {X 0,Y 537.59,Z 194.198,A -85,B 0,C 180,E1 25181.117,E2 25181.117} C_VEL
LIN {X 0,Y 537.543,Z 194.193,A -85,B 0,C 180,E1 25177.851,E2 25177.851} C_VEL
LIN {X 0,Y 537.533,Z 194.2,A -85,B 0,C 180,E1 25174.428,E2 25174.428} C_VEL
LIN {X 0,Y 537.579,Z 194.149,A -85,B 0,C 180,E1 25171.156,E2 25171.156} C_VEL
LIN {X 0,Y 537.545,Z 194.208,A -85,B 0,C 180,E1 25167.986,E2 25167.986} C_VEL
LIN {X 0,Y 537.53,Z 194.181,A -85,B 0,C 180,E1 25164.551,E2 25164.551} C_VEL
LIN {X 0,Y 537.593,Z 194.19,A -85,B 0,C 180,E1 25161.322,E2 25161.322} C_VEL
LIN {X 0,Y 537.546,Z 194.208,A -85,B 0,C 180,E1 25158.068,E2 25158.068} C_VEL
LIN {X 0,Y 537.533,Z 194.198,A -85,B 0,C 180,E1 25154.671,E2 25154.671} C_VEL
LIN {X 0,Y 537.593,Z 194.188,A -85,B 0,C 180,E1 25151.448,E2 25151.448} C_VEL
LIN {X 0,Y 537.584,Z 194.542,A -85,B 0,C 180,E1 25150.407,E2 25150.407} C_VEL
LIN {X 0,Y 543.667,Z 212.614,A -85,B 0,C 180,E1 25147.736,E2 25147.736} C_VEL
LIN {X 0,Y 546.413,Z 221.201,A -85,B 0,C 180,E1 25146.55,E2 25146.55} C_VEL
LIN {X 0,Y 558.786,Z 245.39,A -85,B 0,C 180,E1 25145.228,E2 25145.228} C_VEL
LIN {X 0,Y 560.385,Z 249.36,A -85,B 0,C 180,E1 25145.052,E2 25145.052} C_VEL
LIN {X 0,Y 564.141,Z 268.305,A -85,B 0,C 180,E1 25144.5,E2 25144.5} C_VEL
LIN {X 0,Y 558.693,Z 522.429,A -85,B 0,C 180,E1 25141.048,E2 25141.048} C_VEL
LIN {X 0,Y 557.903,Z 539.952,A -85,B 0,C 180,E1 25140.716,E2 25140.716} C_VEL
LIN {X 0,Y 556.854,Z 557.133,A -85,B 0,C 180,E1 25140.277,E2 25140.277} C_VEL
LIN {X 0,Y 555.605,Z 574.198,A -85,B 0,C 180,E1 25139.722,E2 25139.722} C_VEL
LIN {X 0,Y 554.01,Z 592.688,A -85,B 0,C 180,E1 25138.982,E2 25138.982} C_VEL
LIN {X 0,Y 551.811,Z 614.915,A -85,B 0,C 180,E1 25137.868,E2 25137.868} C_VEL
LIN {X 0,Y 549.952,Z 631.632,A -85,B 0,C 180,E1 25136.856,E2 25136.856} C_VEL
LIN {X 0,Y 548.16,Z 646.908,A -85,B 0,C 180,E1 25135.784,E2 25135.784} C_VEL
LIN {X 0,Y 546.436,Z 661.001,A -85,B 0,C 180,E1 25134.655,E2 25134.655} C_VEL
LIN {X 0,Y 544.714,Z 674.859,A -85,B 0,C 180,E1 25133.391,E2 25133.391} C_VEL
LIN {X 0,Y 543.058,Z 688.255,A -85,B 0,C 180,E1 25132.002,E2 25132.002} C_VEL
LIN {X 0,Y 541.221,Z 703.477,A -85,B 0,C 180,E1 25130.195,E2 25130.195} C_VEL
LIN {X 0,Y 539.61,Z 717.251,A -85,B 0,C 180,E1 25128.247,E2 25128.247} C_VEL
LIN {X 0,Y 538.547,Z 727.308,A -85,B 0,C 180,E1 25126.612,E2 25126.612} C_VEL
LIN {X 0,Y 537.707,Z 736.103,A -85,B 0,C 180,E1 25124.978,E2 25124.978} C_VEL
LIN {X 0,Y 537.038,Z 744.225,A -85,B 0,C 180,E1 25123.237,E2 25123.237} C_VEL
LIN {X 0,Y 536.558,Z 751.164,A -85,B 0,C 180,E1 25121.5,E2 25121.5} C_VEL
LIN {X 0,Y 536.244,Z 757.002,A -85,B 0,C 180,E1 25119.768,E2 25119.768} C_VEL
LIN {X 0,Y 536.051,Z 762.076,A -85,B 0,C 180,E1 25117.933,E2 25117.933} C_VEL
LIN {X 0,Y 535.966,Z 766.076,A -85,B 0,C 180,E1 25116.087,E2 25116.087} C_VEL
LIN {X 0,Y 535.928,Z 769.244,A -85,B 0,C 180,E1 25114.065,E2 25114.065} C_VEL
LIN {X 0,Y 535.919,Z 771.415,A -85,B 0,C 180,E1 25111.603,E2 25111.603} C_VEL
LIN {X 0,Y 535.92,Z 771.708,A -85,B 0,C 180,E1 25109.466,E2 25109.466} C_VEL
LIN {X 0,Y 535.922,Z 770.821,A -85,B 0,C 180,E1 25107.541,E2 25107.541} C_VEL
LIN {X 0,Y 535.93,Z 768.802,A -85,B 0,C 180,E1 25105.614,E2 25105.614} C_VEL
LIN {X 0,Y 535.971,Z 765.837,A -85,B 0,C 180,E1 25103.789,E2 25103.789} C_VEL
LIN {X 0,Y 536.059,Z 761.807,A -85,B 0,C 180,E1 25101.959,E2 25101.959} C_VEL
LIN {X 0,Y 536.259,Z 756.669,A -85,B 0,C 180,E1 25100.124,E2 25100.124} C_VEL
LIN {X 0,Y 536.607,Z 750.365,A -85,B 0,C 180,E1 25098.283,E2 25098.283} C_VEL
LIN {X 0,Y 537.185,Z 742.315,A -85,B 0,C 180,E1 25096.32,E2 25096.32} C_VEL
LIN {X 0,Y 538.247,Z 730.401,A -85,B 0,C 180,E1 25093.933,E2 25093.933} C_VEL
LIN {X 0,Y 539.303,Z 720.058,A -85,B 0,C 180,E1 25092.189,E2 25092.189} C_VEL
LIN {X 0,Y 540.546,Z 708.949,A -85,B 0,C 180,E1 25090.554,E2 25090.554} C_VEL
LIN {X 0,Y 541.849,Z 698.045,A -85,B 0,C 180,E1 25089.139,E2 25089.139} C_VEL
LIN {X 0,Y 543.419,Z 685.256,A -85,B 0,C 180,E1 25087.672,E2 25087.672} C_VEL
LIN {X 0,Y 545.233,Z 670.834,A -85,B 0,C 180,E1 25086.221,E2 25086.221} C_VEL
LIN {X 0,Y 547.683,Z 650.934,A -85,B 0,C 180,E1 25084.52,E2 25084.52} C_VEL
LIN {X 0,Y 549.577,Z 634.857,A -85,B 0,C 180,E1 25083.358,E2 25083.358} C_VEL
LIN {X 0,Y 551.292,Z 619.519,A -85,B 0,C 180,E1 25082.397,E2 25082.397} C_VEL
LIN {X 0,Y 552.936,Z 603.788,A -85,B 0,C 180,E1 25081.548,E2 25081.548} C_VEL
LIN {X 0,Y 554.469,Z 587.585,A -85,B 0,C 180,E1 25080.802,E2 25080.802} C_VEL
LIN {X 0,Y 555.834,Z 571.326,A -85,B 0,C 180,E1 25080.177,E2 25080.177} C_VEL
LIN {X 0,Y 557.064,Z 554.098,A -85,B 0,C 180,E1 25079.637,E2 25079.637} C_VEL
LIN {X 0,Y 558.184,Z 534.961,A -85,B 0,C 180,E1 25079.175,E2 25079.175} C_VEL
LIN {X 0,Y 559.132,Z 505.855,A -85,B 0,C 180,E1 25078.71,E2 25078.71} C_VEL
LIN {X 0,Y 564.082,Z 267.05,A -85,B 0,C 180,E1 25075.477,E2 25075.477} C_VEL
LIN {X 0,Y 559.765,Z 247.461,A -85,B 0,C 180,E1 25074.874,E2 25074.874} C_VEL
LIN {X 0,Y 550.125,Z 228.541,A -85,B 0,C 180,E1 25073.871,E2 25073.871} C_VEL
LIN {X 0,Y 546.272,Z 220.806,A -85,B 0,C 180,E1 25073.415,E2 25073.415} C_VEL
LIN {X 0,Y 540.398,Z 202.703,A -85,B 0,C 180,E1 25070.83,E2 25070.83} C_VEL
LIN {X 0,Y 537.547,Z 194.309,A -85,B 0,C 180,E1 25069.527,E2 25069.527} C_VEL
LIN {X 0,Y 537.588,Z 194.205,A -85,B 0,C 180,E1 25066.346,E2 25066.346} C_VEL
LIN {X 0,Y 537.55,Z 194.201,A -85,B 0,C 180,E1 25063.037,E2 25063.037} C_VEL
LIN {X 0,Y 537.532,Z 194.183,A -85,B 0,C 180,E1 25059.784,E2 25059.784} C_VEL
LIN {X 0,Y 537.592,Z 194.194,A -85,B 0,C 180,E1 25056.659,E2 25056.659} C_VEL
LIN {X 0,Y 537.536,Z 194.198,A -85,B 0,C 180,E1 25053.375,E2 25053.375} C_VEL
LIN {X 0,Y 537.533,Z 194.179,A -85,B 0,C 180,E1 25049.902,E2 25049.902} C_VEL
LIN {X 0,Y 537.59,Z 194.165,A -85,B 0,C 180,E1 25046.751,E2 25046.751} C_VEL
LIN {X 0,Y 537.539,Z 194.207,A -85,B 0,C 180,E1 25043.458,E2 25043.458} C_VEL
LIN {X 0,Y 537.536,Z 194.207,A -85,B 0,C 180,E1 25040.015,E2 25040.015} C_VEL
LIN {X 0,Y 537.591,Z 194.19,A -85,B 0,C 180,E1 25036.716,E2 25036.716} C_VEL
LIN {X 0,Y 537.537,Z 194.197,A -85,B 0,C 180,E1 25033.555,E2 25033.555} C_VEL
LIN {X 0,Y 537.534,Z 194.205,A -85,B 0,C 180,E1 25030.07,E2 25030.07} C_VEL
LIN {X 0,Y 537.596,Z 194.192,A -85,B 0,C 180,E1 25026.837,E2 25026.837} C_VEL
LIN {X 0,Y 537.544,Z 194.196,A -85,B 0,C 180,E1 25023.519,E2 25023.519} C_VEL
LIN {X 0,Y 537.533,Z 194.208,A -85,B 0,C 180,E1 25020.213,E2 25020.213} C_VEL
LIN {X 0,Y 537.589,Z 194.189,A -85,B 0,C 180,E1 25017.015,E2 25017.015} C_VEL
LIN {X 0,Y 537.534,Z 194.203,A -85,B 0,C 180,E1 25013.806,E2 25013.806} C_VEL
LIN {X 0,Y 537.536,Z 194.208,A -85,B 0,C 180,E1 25010.311,E2 25010.311} C_VEL
LIN {X 0,Y 537.586,Z 194.192,A -85,B 0,C 180,E1 25006.994,E2 25006.994} C_VEL
LIN {X 0,Y 537.54,Z 194.201,A -85,B 0,C 180,E1 25003.798,E2 25003.798} C_VEL
LIN {X 0,Y 537.535,Z 194.207,A -85,B 0,C 180,E1 25000.438,E2 25000.438} C_VEL
LIN {X 0,Y 537.604,Z 194.196,A -85,B 0,C 180,E1 24997.241,E2 24997.241} C_VEL
LIN {X 0,Y 537.537,Z 194.175,A -85,B 0,C 180,E1 24993.938,E2 24993.938} C_VEL
LIN {X 0,Y 537.53,Z 194.178,A -85,B 0,C 180,E1 24990.509,E2 24990.509} C_VEL
LIN {X 0,Y 537.593,Z 194.195,A -85,B 0,C 180,E1 24987.358,E2 24987.358} C_VEL
LIN {X 0,Y 537.537,Z 194.167,A -85,B 0,C 180,E1 24983.999,E2 24983.999} C_VEL
LIN {X 0,Y 537.534,Z 194.21,A -85,B 0,C 180,E1 24980.631,E2 24980.631} C_VEL
LIN {X 0,Y 537.59,Z 194.207,A -85,B 0,C 180,E1 24977.388,E2 24977.388} C_VEL
LIN {X 0,Y 537.546,Z 194.211,A -85,B 0,C 180,E1 24974.074,E2 24974.074} C_VEL
LIN {X 0,Y 537.536,Z 194.208,A -85,B 0,C 180,E1 24970.754,E2 24970.754} C_VEL
LIN {X 0,Y 537.596,Z 194.203,A -85,B 0,C 180,E1 24967.588,E2 24967.588} C_VEL
LIN {X 0,Y 537.54,Z 194.211,A -85,B 0,C 180,E1 24964.301,E2 24964.301} C_VEL
LIN {X 0,Y 537.534,Z 194.209,A -85,B 0,C 180,E1 24960.886,E2 24960.886} C_VEL
LIN {X 0,Y 537.602,Z 194.202,A -85,B 0,C 180,E1 24957.705,E2 24957.705} C_VEL
LIN {X 0,Y 537.541,Z 194.212,A -85,B 0,C 180,E1 24954.387,E2 24954.387} C_VEL
LIN {X 0,Y 537.534,Z 194.21,A -85,B 0,C 180,E1 24950.966,E2 24950.966} C_VEL
LIN {X 0,Y 537.593,Z 194.206,A -85,B 0,C 180,E1 24947.757,E2 24947.757} C_VEL
LIN {X 0,Y 537.579,Z 194.513,A -85,B 0,C 180,E1 24945.092,E2 24945.092} C_VEL
LIN {X 0,Y 538.067,Z 196.164,A -85,B 0,C 180,E1 24944.142,E2 24944.142} C_VEL
LIN {X 0,Y 539.34,Z 198.358,A -85,B 0,C 180,E1 24943.07,E2 24943.07} C_VEL
LIN {X 0,Y 541.564,Z 200.2,A -85,B 0,C 180,E1 24941.177,E2 24941.177} C_VEL
LIN {X 0,Y 543.957,Z 201.477,A -85,B 0,C 180,E1 24938.775,E2 24938.775} C_VEL
LIN {X 0,Y 544.962,Z 203.146,A -85,B 0,C 180,E1 24937.378,E2 24937.378} C_VEL
LIN {X 0,Y 545.966,Z 204.868,A -85,B 0,C 180,E1 24935.675,E2 24935.675} C_VEL
LIN {X 0,Y 546.974,Z 206.021,A -85,B 0,C 180,E1 24933.248,E2 24933.248} C_VEL
LIN {X 0,Y 547.46,Z 206.435,A -85,B 0,C 180,E1 24930.732,E2 24930.732} C_VEL
LIN {X 0,Y 547.497,Z 206.44,A -85,B 0,C 180,E1 24930.337,E2 24930.337} C_VEL
LIN {X 0,Y 547.421,Z 207.426,A -85,B 0,C 180,E1 24929.53,E2 24929.53} C_VEL
LIN {X 0,Y 546.341,Z 213.303,A -85,B 0,C 180,E1 24927.454,E2 24927.454} C_VEL
LIN {X 0,Y 545.982,Z 213.947,A -85,B 0,C 180,E1 24926.702,E2 24926.702} C_VEL
LIN {X 0,Y 544.915,Z 212.727,A -85,B 0,C 180,E1 24924.209,E2 24924.209} C_VEL
LIN {X 0,Y 543.9,Z 210.993,A -85,B 0,C 180,E1 24922.501,E2 24922.501} C_VEL
LIN {X 0,Y 542.872,Z 209.345,A -85,B 0,C 180,E1 24921.101,E2 24921.101} C_VEL
LIN {X 0,Y 540.295,Z 207.976,A -85,B 0,C 180,E1 24918.581,E2 24918.581} C_VEL
LIN {X 0,Y 538.065,Z 206.008,A -85,B 0,C 180,E1 24916.68,E2 24916.68} C_VEL
LIN {X 0,Y 535.765,Z 202.297,A -85,B 0,C 180,E1 24914.856,E2 24914.856} C_VEL
LIN {X 0,Y 532.218,Z 200.167,A -85,B 0,C 180,E1 24912.63,E2 24912.63} C_VEL
LIN {X 0,Y 530.164,Z 197.325,A -85,B 0,C 180,E1 24911.359,E2 24911.359} C_VEL
LIN {X 0,Y 529.675,Z 195.622,A -85,B 0,C 180,E1 24910.712,E2 24910.712} C_VEL
LIN {X 0,Y 529.595,Z 195.201,A -85,B 0,C 180,E1 24909.444,E2 24909.444} C_VEL
LIN {X 0,Y 529.653,Z 195.192,A -85,B 0,C 180,E1 24906.175,E2 24906.175} C_VEL
LIN {X 0,Y 529.612,Z 195.199,A -85,B 0,C 180,E1 24902.818,E2 24902.818} C_VEL
LIN {X 0,Y 529.593,Z 195.199,A -85,B 0,C 180,E1 24899.482,E2 24899.482} C_VEL
LIN {X 0,Y 529.638,Z 195.194,A -85,B 0,C 180,E1 24896.162,E2 24896.162} C_VEL
LIN {X 0,Y 529.621,Z 195.199,A -85,B 0,C 180,E1 24892.817,E2 24892.817} C_VEL
LIN {X 0,Y 529.594,Z 195.198,A -85,B 0,C 180,E1 24889.504,E2 24889.504} C_VEL
LIN {X 0,Y 529.641,Z 195.194,A -85,B 0,C 180,E1 24886.302,E2 24886.302} C_VEL
LIN {X 0,Y 529.618,Z 195.198,A -85,B 0,C 180,E1 24882.965,E2 24882.965} C_VEL
LIN {X 0,Y 529.592,Z 195.199,A -85,B 0,C 180,E1 24879.627,E2 24879.627} C_VEL
LIN {X 0,Y 529.63,Z 195.157,A -85,B 0,C 180,E1 24876.356,E2 24876.356} C_VEL
LIN {X 0,Y 529.617,Z 195.181,A -85,B 0,C 180,E1 24873.056,E2 24873.056} C_VEL
LIN {X 0,Y 529.59,Z 195.172,A -85,B 0,C 180,E1 24869.729,E2 24869.729} C_VEL
LIN {X 0,Y 529.63,Z 195.145,A -85,B 0,C 180,E1 24866.458,E2 24866.458} C_VEL
LIN {X 0,Y 529.618,Z 195.198,A -85,B 0,C 180,E1 24863.176,E2 24863.176} C_VEL
LIN {X 0,Y 529.592,Z 195.196,A -85,B 0,C 180,E1 24859.868,E2 24859.868} C_VEL
LIN {X 0,Y 529.633,Z 195.179,A -85,B 0,C 180,E1 24856.563,E2 24856.563} C_VEL
LIN {X 0,Y 529.605,Z 195.192,A -85,B 0,C 180,E1 24853.428,E2 24853.428} C_VEL
LIN {X 0,Y 529.593,Z 195.196,A -85,B 0,C 180,E1 24850.003,E2 24850.003} C_VEL
LIN {X 0,Y 529.639,Z 195.178,A -85,B 0,C 180,E1 24846.722,E2 24846.722} C_VEL
LIN {X 0,Y 529.61,Z 195.192,A -85,B 0,C 180,E1 24843.464,E2 24843.464} C_VEL
LIN {X 0,Y 529.591,Z 195.196,A -85,B 0,C 180,E1 24840.108,E2 24840.108} C_VEL
LIN {X 0,Y 529.639,Z 195.175,A -85,B 0,C 180,E1 24836.862,E2 24836.862} C_VEL
LIN {X 0,Y 529.611,Z 195.194,A -85,B 0,C 180,E1 24833.604,E2 24833.604} C_VEL
LIN {X 0,Y 529.593,Z 195.194,A -85,B 0,C 180,E1 24830.204,E2 24830.204} C_VEL
LIN {X 0,Y 529.635,Z 195.178,A -85,B 0,C 180,E1 24826.906,E2 24826.906} C_VEL
LIN {X 0,Y 529.606,Z 195.196,A -85,B 0,C 180,E1 24823.774,E2 24823.774} C_VEL
LIN {X 0,Y 529.594,Z 195.197,A -85,B 0,C 180,E1 24820.362,E2 24820.362} C_VEL
LIN {X 0,Y 529.646,Z 195.183,A -85,B 0,C 180,E1 24817.094,E2 24817.094} C_VEL
LIN {X 0,Y 529.611,Z 195.17,A -85,B 0,C 180,E1 24813.782,E2 24813.782} C_VEL
LIN {X 0,Y 529.59,Z 195.155,A -85,B 0,C 180,E1 24810.476,E2 24810.476} C_VEL
LIN {X 0,Y 529.653,Z 195.188,A -85,B 0,C 180,E1 24807.322,E2 24807.322} C_VEL
LIN {X 0,Y 529.612,Z 195.177,A -85,B 0,C 180,E1 24803.91,E2 24803.91} C_VEL
LIN {X 0,Y 529.59,Z 195.174,A -85,B 0,C 180,E1 24800.543,E2 24800.543} C_VEL
LIN {X 0,Y 529.638,Z 195.19,A -85,B 0,C 180,E1 24797.247,E2 24797.247} C_VEL
LIN {X 0,Y 529.615,Z 195.198,A -85,B 0,C 180,E1 24794.001,E2 24794.001} C_VEL
LIN {X 0,Y 529.633,Z 195.355,A -85,B 0,C 180,E1 24791.028,E2 24791.028} C_VEL
LIN {X 0,Y 535.551,Z 212.77,A -85,B 0,C 180,E1 24788.357,E2 24788.357} C_VEL
LIN {X 0,Y 538.053,Z 220.782,A -85,B 0,C 180,E1 24787.221,E2 24787.221} C_VEL
LIN {X 0,Y 550.664,Z 244.958,A -85,B 0,C 180,E1 24785.83,E2 24785.83} C_VEL
LIN {X 0,Y 554.179,Z 252.721,A -85,B 0,C 180,E1 24785.449,E2 24785.449} C_VEL
LIN {X 0,Y 557.509,Z 269.807,A -85,B 0,C 180,E1 24784.944,E2 24784.944} C_VEL
LIN {X 0,Y 551.829,Z 522.562,A -85,B 0,C 180,E1 24781.472,E2 24781.472} C_VEL
LIN {X 0,Y 551.002,Z 540.095,A -85,B 0,C 180,E1 24781.135,E2 24781.135} C_VEL
LIN {X 0,Y 549.903,Z 557.332,A -85,B 0,C 180,E1 24780.689,E2 24780.689} C_VEL
LIN {X 0,Y 548.498,Z 575.611,A -85,B 0,C 180,E1 24780.082,E2 24780.082} C_VEL
LIN {X 0,Y 546.519,Z 597.236,A -85,B 0,C 180,E1 24779.177,E2 24779.177} C_VEL
LIN {X 0,Y 544.494,Z 616.203,A -85,B 0,C 180,E1 24778.181,E2 24778.181} C_VEL
LIN {X 0,Y 542.723,Z 631.455,A -85,B 0,C 180,E1 24777.243,E2 24777.243} C_VEL
LIN {X 0,Y 540.885,Z 646.461,A -85,B 0,C 180,E1 24776.179,E2 24776.179} C_VEL
LIN {X 0,Y 539.043,Z 660.823,A -85,B 0,C 180,E1 24775.016,E2 24775.016} C_VEL
LIN {X 0,Y 537.259,Z 674.463,A -85,B 0,C 180,E1 24773.758,E2 24773.758} C_VEL
LIN {X 0,Y 535.549,Z 687.576,A -85,B 0,C 180,E1 24772.385,E2 24772.385} C_VEL
LIN {X 0,Y 533.771,Z 701.427,A -85,B 0,C 180,E1 24770.732,E2 24770.732} C_VEL
LIN {X 0,Y 531.938,Z 716.371,A -85,B 0,C 180,E1 24768.633,E2 24768.633} C_VEL
LIN {X 0,Y 530.708,Z 727.258,A -85,B 0,C 180,E1 24766.841,E2 24766.841} C_VEL
LIN {X 0,Y 529.834,Z 735.924,A -85,B 0,C 180,E1 24765.205,E2 24765.205} C_VEL
LIN {X 0,Y 529.114,Z 744.047,A -85,B 0,C 180,E1 24763.439,E2 24763.439} C_VEL
LIN {X 0,Y 528.603,Z 750.986,A -85,B 0,C 180,E1 24761.676,E2 24761.676} C_VEL
LIN {X 0,Y 528.268,Z 756.825,A -85,B 0,C 180,E1 24759.917,E2 24759.917} C_VEL
LIN {X 0,Y 528.061,Z 761.9,A -85,B 0,C 180,E1 24758.054,E2 24758.054} C_VEL
LIN {X 0,Y 527.968,Z 765.989,A -85,B 0,C 180,E1 24756.133,E2 24756.133} C_VEL
LIN {X 0,Y 527.928,Z 769.216,A -85,B 0,C 180,E1 24754.018,E2 24754.018} C_VEL
LIN {X 0,Y 527.919,Z 771.269,A -85,B 0,C 180,E1 24751.519,E2 24751.519} C_VEL
LIN {X 0,Y 527.922,Z 771.534,A -85,B 0,C 180,E1 24749.457,E2 24749.457} C_VEL
LIN {X 0,Y 527.923,Z 770.646,A -85,B 0,C 180,E1 24747.504,E2 24747.504} C_VEL
LIN {X 0,Y 527.93,Z 768.774,A -85,B 0,C 180,E1 24745.656,E2 24745.656} C_VEL
LIN {X 0,Y 527.97,Z 765.869,A -85,B 0,C 180,E1 24743.804,E2 24743.804} C_VEL
LIN {X 0,Y 528.061,Z 761.9,A -85,B 0,C 180,E1 24741.946,E2 24741.946} C_VEL
LIN {X 0,Y 528.268,Z 756.825,A -85,B 0,C 180,E1 24740.083,E2 24740.083} C_VEL
LIN {X 0,Y 528.603,Z 750.986,A -85,B 0,C 180,E1 24738.324,E2 24738.324} C_VEL
LIN {X 0,Y 529.114,Z 744.047,A -85,B 0,C 180,E1 24736.561,E2 24736.561} C_VEL
LIN {X 0,Y 529.834,Z 735.924,A -85,B 0,C 180,E1 24734.795,E2 24734.795} C_VEL
LIN {X 0,Y 530.789,Z 726.51,A -85,B 0,C 180,E1 24733.025,E2 24733.025} C_VEL
LIN {X 0,Y 532.296,Z 713.52,A -85,B 0,C 180,E1 24730.925,E2 24730.925} C_VEL
LIN {X 0,Y 533.991,Z 699.647,A -85,B 0,C 180,E1 24729.047,E2 24729.047} C_VEL
LIN {X 0,Y 535.658,Z 686.695,A -85,B 0,C 180,E1 24727.518,E2 24727.518} C_VEL
LIN {X 0,Y 537.333,Z 673.902,A -85,B 0,C 180,E1 24726.187,E2 24726.187} C_VEL
LIN {X 0,Y 539.105,Z 660.357,A -85,B 0,C 180,E1 24724.944,E2 24724.944} C_VEL
LIN {X 0,Y 540.944,Z 646.018,A -85,B 0,C 180,E1 24723.787,E2 24723.787} C_VEL
LIN {X 0,Y 542.921,Z 629.842,A -85,B 0,C 180,E1 24722.649,E2 24722.649} C_VEL
LIN {X 0,Y 545.301,Z 608.925,A -85,B 0,C 180,E1 24721.411,E2 24721.411} C_VEL
LIN {X 0,Y 547.194,Z 590.022,A -85,B 0,C 180,E1 24720.502,E2 24720.502} C_VEL
LIN {X 0,Y 548.663,Z 573.588,A -85,B 0,C 180,E1 24719.845,E2 24719.845} C_VEL
LIN {X 0,Y 549.974,Z 556.325,A -85,B 0,C 180,E1 24719.282,E2 24719.282} C_VEL
LIN {X 0,Y 551.041,Z 539.4,A -85,B 0,C 180,E1 24718.85,E2 24718.85} C_VEL
LIN {X 0,Y 551.853,Z 521.841,A -85,B 0,C 180,E1 24718.516,E2 24718.516} C_VEL
LIN {X 0,Y 557.528,Z 269.022,A -85,B 0,C 180,E1 24715.045,E2 24715.045} C_VEL
LIN {X 0,Y 553.677,Z 251.176,A -85,B 0,C 180,E1 24714.49,E2 24714.49} C_VEL
LIN {X 0,Y 542.867,Z 229.929,A -85,B 0,C 180,E1 24713.335,E2 24713.335} C_VEL
LIN {X 0,Y 538.052,Z 220.782,A -85,B 0,C 180,E1 24712.779,E2 24712.779} C_VEL
LIN {X 0,Y 532.292,Z 203.116,A -85,B 0,C 180,E1 24710.201,E2 24710.201} C_VEL
LIN {X 0,Y 529.629,Z 195.317,A -85,B 0,C 180,E1 24708.959,E2 24708.959} C_VEL
LIN {X 0,Y 529.594,Z 195.191,A -85,B 0,C 180,E1 24705.544,E2 24705.544} C_VEL
LIN {X 0,Y 529.633,Z 195.197,A -85,B 0,C 180,E1 24702.229,E2 24702.229} C_VEL
LIN {X 0,Y 529.622,Z 195.179,A -85,B 0,C 180,E1 24698.948,E2 24698.948} C_VEL
LIN {X 0,Y 529.591,Z 195.172,A -85,B 0,C 180,E1 24695.691,E2 24695.691} C_VEL
LIN {X 0,Y 529.643,Z 195.195,A -85,B 0,C 180,E1 24692.422,E2 24692.422} C_VEL
LIN {X 0,Y 529.6,Z 195.148,A -85,B 0,C 180,E1 24689.275,E2 24689.275} C_VEL
LIN {X 0,Y 529.594,Z 195.184,A -85,B 0,C 180,E1 24685.858,E2 24685.858} C_VEL
LIN {X 0,Y 529.64,Z 195.178,A -85,B 0,C 180,E1 24682.535,E2 24682.535} C_VEL
LIN {X 0,Y 529.612,Z 195.195,A -85,B 0,C 180,E1 24679.291,E2 24679.291} C_VEL
LIN {X 0,Y 529.593,Z 195.193,A -85,B 0,C 180,E1 24675.889,E2 24675.889} C_VEL
LIN {X 0,Y 529.634,Z 195.176,A -85,B 0,C 180,E1 24672.603,E2 24672.603} C_VEL
LIN {X 0,Y 529.617,Z 195.191,A -85,B 0,C 180,E1 24669.344,E2 24669.344} C_VEL
LIN {X 0,Y 529.593,Z 195.196,A -85,B 0,C 180,E1 24666.069,E2 24666.069} C_VEL
LIN {X 0,Y 529.642,Z 195.176,A -85,B 0,C 180,E1 24662.814,E2 24662.814} C_VEL
LIN {X 0,Y 529.605,Z 195.197,A -85,B 0,C 180,E1 24659.567,E2 24659.567} C_VEL
LIN {X 0,Y 529.593,Z 195.195,A -85,B 0,C 180,E1 24656.211,E2 24656.211} C_VEL
LIN {X 0,Y 529.65,Z 195.175,A -85,B 0,C 180,E1 24652.952,E2 24652.952} C_VEL
LIN {X 0,Y 529.608,Z 195.197,A -85,B 0,C 180,E1 24649.668,E2 24649.668} C_VEL
LIN {X 0,Y 529.591,Z 195.195,A -85,B 0,C 180,E1 24646.238,E2 24646.238} C_VEL
LIN {X 0,Y 529.639,Z 195.178,A -85,B 0,C 180,E1 24642.985,E2 24642.985} C_VEL
LIN {X 0,Y 529.616,Z 195.193,A -85,B 0,C 180,E1 24639.673,E2 24639.673} C_VEL
LIN {X 0,Y 529.595,Z 195.198,A -85,B 0,C 180,E1 24636.405,E2 24636.405} C_VEL
LIN {X 0,Y 529.644,Z 195.137,A -85,B 0,C 180,E1 24633.179,E2 24633.179} C_VEL
LIN {X 0,Y 529.6,Z 195.182,A -85,B 0,C 180,E1 24629.979,E2 24629.979} C_VEL
LIN {X 0,Y 529.592,Z 195.176,A -85,B 0,C 180,E1 24626.543,E2 24626.543} C_VEL
LIN {X 0,Y 529.64,Z 195.166,A -85,B 0,C 180,E1 24623.241,E2 24623.241} C_VEL
LIN {X 0,Y 529.605,Z 195.198,A -85,B 0,C 180,E1 24620.033,E2 24620.033} C_VEL
LIN {X 0,Y 529.594,Z 195.199,A -85,B 0,C 180,E1 24616.587,E2 24616.587} C_VEL
LIN {X 0,Y 529.634,Z 195.196,A -85,B 0,C 180,E1 24613.252,E2 24613.252} C_VEL
LIN {X 0,Y 529.62,Z 195.198,A -85,B 0,C 180,E1 24609.959,E2 24609.959} C_VEL
LIN {X 0,Y 529.594,Z 195.198,A -85,B 0,C 180,E1 24606.622,E2 24606.622} C_VEL
LIN {X 0,Y 529.623,Z 195.197,A -85,B 0,C 180,E1 24603.243,E2 24603.243} C_VEL
LIN {X 0,Y 529.623,Z 195.199,A -85,B 0,C 180,E1 24600.015,E2 24600.015} C_VEL
LIN {X 0,Y 529.593,Z 195.198,A -85,B 0,C 180,E1 24596.698,E2 24596.698} C_VEL
LIN {X 0,Y 529.622,Z 195.198,A -85,B 0,C 180,E1 24593.354,E2 24593.354} C_VEL
LIN {X 0,Y 529.616,Z 195.198,A -85,B 0,C 180,E1 24590.209,E2 24590.209} C_VEL
LIN {X 0,Y 529.676,Z 195.622,A -85,B 0,C 180,E1 24589.287,E2 24589.287} C_VEL
LIN {X 0,Y 530.432,Z 197.879,A -85,B 0,C 180,E1 24588.46,E2 24588.46} C_VEL
LIN {X 0,Y 532.584,Z 200.49,A -85,B 0,C 180,E1 24587.134,E2 24587.134} C_VEL
LIN {X 0,Y 536.122,Z 202.637,A -85,B 0,C 180,E1 24584.912,E2 24584.912} C_VEL
LIN {X 0,Y 538.19,Z 206.172,A -85,B 0,C 180,E1 24583.208,E2 24583.208} C_VEL
LIN {X 0,Y 540.428,Z 208.062,A -85,B 0,C 180,E1 24581.304,E2 24581.304} C_VEL
LIN {X 0,Y 542.872,Z 209.345,A -85,B 0,C 180,E1 24578.899,E2 24578.899} C_VEL
LIN {X 0,Y 543.9,Z 210.992,A -85,B 0,C 180,E1 24577.499,E2 24577.499} C_VEL
LIN {X 0,Y 544.915,Z 212.728,A -85,B 0,C 180,E1 24575.791,E2 24575.791} C_VEL
LIN {X 0,Y 545.962,Z 213.925,A -85,B 0,C 180,E1 24573.359,E2 24573.359} C_VEL
LIN {X 0,Y 546.479,Z 214.375,A -85,B 0,C 180,E1 24570.839,E2 24570.839} C_VEL
LIN {X 0,Y 546.392,Z 214.279,A -85,B 0,C 180,E1 24568.322,E2 24568.322} C_VEL
LIN {X 0,Y 545.982,Z 213.947,A -85,B 0,C 180,E1 24566.702,E2 24566.702} C_VEL
LIN {X 0,Y 545.707,Z 214.778,A -85,B 0,C 180,E1 24566.158,E2 24566.158} C_VEL
LIN {X 0,Y 544.407,Z 220.188,A -85,B 0,C 180,E1 24564.836,E2 24564.836} C_VEL
LIN {X 0,Y 543.982,Z 220.78,A -85,B 0,C 180,E1 24564.293,E2 24564.293} C_VEL
